    movel([0.070135, -1.347885, -2.596834, -0.767670, 1.570796, 1.640931],accel_mss,speed_ms,0,blend_radius_m)
    movel([0.070293, -1.348064, -2.596716, -0.767609, 1.570796, 1.641090],accel_mss,speed_ms,0,blend_radius_m)
    movel([0.070585, -1.348016, -2.596748, -0.767625, 1.570796, 1.641381],accel_mss,speed_ms,0,blend_radius_m)
    movel([0.071041, -1.347896, -2.596827, -0.767666, 1.570796, 1.641837],accel_mss,speed_ms,0,blend_radius_m)
    movel([0.071762, -1.347670, -2.596975, -0.767743, 1.570796, 1.642559],accel_mss,speed_ms,0,blend_radius_m)
    movel([0.072728, -1.347369, -2.597173, -0.767846, 1.570796, 1.643524],accel_mss,speed_ms,0,blend_radius_m)
    movel([0.073151, -1.347276, -2.597235, -0.767878, 1.570796, 1.643947],accel_mss,speed_ms,0,blend_radius_m)
    movel([0.073323, -1.347462, -2.597113, -0.767815, 1.570796, 1.644120],accel_mss,speed_ms,0,blend_radius_m)
    movel([0.072183, -1.349035, -2.596076, -0.767279, 1.570796, 1.642979],accel_mss,speed_ms,0,blend_radius_m)
    movel([0.070974, -1.350670, -2.594994, -0.766725, 1.570796, 1.641770],accel_mss,speed_ms,0,blend_radius_m)
    movel([0.069560, -1.352574, -2.593730, -0.766085, 1.570796, 1.640356],accel_mss,speed_ms,0,blend_radius_m)
    movel([0.068144, -1.354467, -2.592468, -0.765453, 1.570796, 1.638941],accel_mss,speed_ms,0,blend_radius_m)
    movel([0.066928, -1.356066, -2.591399, -0.764924, 1.570796, 1.637725],accel_mss,speed_ms,0,blend_radius_m)
    movel([0.065852, -1.357467, -2.590459, -0.764463, 1.570796, 1.636649],accel_mss,speed_ms,0,blend_radius_m)
    speed_ms = 0.003
    movel([0.065746, -1.344239, -2.584239, -0.783911, 1.570796, 1.636542],accel_mss,speed_ms,0,blend_radius_m)
    speed_ms = 1.000
    movel([0.065746, -1.318776, -2.571512, -0.822101, 1.570796, 1.636542],accel_mss,speed_ms,0,blend_radius_m)
    movel([0.081492, -1.289170, -2.589753, -0.833466, 1.570796, 1.652288],accel_mss,speed_ms,0,blend_radius_m)
    movel([0.081492, -1.315103, -2.602865, -0.794421, 1.570796, 1.652288],accel_mss,speed_ms,0,blend_radius_m)
    speed_ms = 0.003
    movel([0.081492, -1.325253, -2.607648, -0.779489, 1.570796, 1.652288],accel_mss,speed_ms,0,blend_radius_m)
    speed_ms = 0.007
    movel([0.081341, -1.325030, -2.607788, -0.779571, 1.570796, 1.652138],accel_mss,speed_ms,0,blend_radius_m)
    movel([0.081467, -1.324183, -2.608320, -0.779886, 1.570796, 1.652263],accel_mss,speed_ms,0,blend_radius_m)
    movel([0.081769, -1.322931, -2.609105, -0.780353, 1.570796, 1.652565],accel_mss,speed_ms,0,blend_radius_m)
    movel([0.082314, -1.321124, -2.610234, -0.781031, 1.570796, 1.653110],accel_mss,speed_ms,0,blend_radius_m)
    movel([0.082603, -1.320135, -2.610851, -0.781404, 1.570796, 1.653400],accel_mss,speed_ms,0,blend_radius_m)
    movel([0.082660, -1.319646, -2.611154, -0.781588, 1.570796, 1.653456],accel_mss,speed_ms,0,blend_radius_m)
    movel([0.082527, -1.319485, -2.611255, -0.781649, 1.570796, 1.653323],accel_mss,speed_ms,0,blend_radius_m)
    movel([0.082236, -1.319545, -2.611217, -0.781627, 1.570796, 1.653033],accel_mss,speed_ms,0,blend_radius_m)
    movel([0.081751, -1.319793, -2.611063, -0.781533, 1.570796, 1.652547],accel_mss,speed_ms,0,blend_radius_m)
    movel([0.081384, -1.319972, -2.610952, -0.781465, 1.570796, 1.652181],accel_mss,speed_ms,0,blend_radius_m)
    movel([0.081002, -1.320156, -2.610837, -0.781396, 1.570796, 1.651798],accel_mss,speed_ms,0,blend_radius_m)
    movel([0.080195, -1.320466, -2.610644, -0.781279, 1.570796, 1.650992],accel_mss,speed_ms,0,blend_radius_m)
    movel([0.079870, -1.320370, -2.610704, -0.781315, 1.570796, 1.650667],accel_mss,speed_ms,0,blend_radius_m)
    movel([0.079791, -1.319865, -2.611018, -0.781506, 1.570796, 1.650588],accel_mss,speed_ms,0,blend_radius_m)
    movel([0.079966, -1.317934, -2.612217, -0.782238, 1.570796, 1.650762],accel_mss,speed_ms,0,blend_radius_m)
    movel([0.080077, -1.316920, -2.612844, -0.782625, 1.570796, 1.650873],accel_mss,speed_ms,0,blend_radius_m)
    movel([0.080182, -1.316146, -2.613323, -0.782921, 1.570796, 1.650979],accel_mss,speed_ms,0,blend_radius_m)
    movel([0.080285, -1.315545, -2.613693, -0.783151, 1.570796, 1.651081],accel_mss,speed_ms,0,blend_radius_m)
    movel([0.080559, -1.315193, -2.613910, -0.783286, 1.570796, 1.651355],accel_mss,speed_ms,0,blend_radius_m)
    movel([0.080916, -1.314988, -2.614036, -0.783365, 1.570796, 1.651713],accel_mss,speed_ms,0,blend_radius_m)
    movel([0.081474, -1.314721, -2.614200, -0.783468, 1.570796, 1.652271],accel_mss,speed_ms,0,blend_radius_m)
    movel([0.082380, -1.314335, -2.614437, -0.783616, 1.570796, 1.653176],accel_mss,speed_ms,0,blend_radius_m)
    movel([0.083212, -1.314002, -2.614642, -0.783745, 1.570796, 1.654008],accel_mss,speed_ms,0,blend_radius_m)
    movel([0.083713, -1.313842, -2.614741, -0.783807, 1.570796, 1.654510],accel_mss,speed_ms,0,blend_radius_m)
    movel([0.084029, -1.313805, -2.614764, -0.783821, 1.570796, 1.654826],accel_mss,speed_ms,0,blend_radius_m)
    movel([0.084275, -1.313954, -2.614672, -0.783763, 1.570796, 1.655071],accel_mss,speed_ms,0,blend_radius_m)
    movel([0.084281, -1.314246, -2.614492, -0.783650, 1.570796, 1.655077],accel_mss,speed_ms,0,blend_radius_m)
    movel([0.084076, -1.314711, -2.614206, -0.783471, 1.570796, 1.654872],accel_mss,speed_ms,0,blend_radius_m)
    movel([0.083648, -1.315836, -2.613514, -0.783039, 1.570796, 1.654444],accel_mss,speed_ms,0,blend_radius_m)
    movel([0.083205, -1.317019, -2.612783, -0.782587, 1.570796, 1.654001],accel_mss,speed_ms,0,blend_radius_m)
    movel([0.083202, -1.317302, -2.612608, -0.782479, 1.570796, 1.653998],accel_mss,speed_ms,0,blend_radius_m)
    movel([0.083652, -1.317193, -2.612675, -0.782520, 1.570796, 1.654448],accel_mss,speed_ms,0,blend_radius_m)
    movel([0.084222, -1.316970, -2.612813, -0.782605, 1.570796, 1.655019],accel_mss,speed_ms,0,blend_radius_m)
    movel([0.084649, -1.316806, -2.612915, -0.782668, 1.570796, 1.655445],accel_mss,speed_ms,0,blend_radius_m)
    movel([0.085028, -1.316673, -2.612997, -0.782719, 1.570796, 1.655825],accel_mss,speed_ms,0,blend_radius_m)
    movel([0.085344, -1.316573, -2.613059, -0.782757, 1.570796, 1.656140],accel_mss,speed_ms,0,blend_radius_m)
    movel([0.085547, -1.316717, -2.612970, -0.782702, 1.570796, 1.656343],accel_mss,speed_ms,0,blend_radius_m)
    movel([0.085460, -1.317124, -2.612719, -0.782547, 1.570796, 1.656257],accel_mss,speed_ms,0,blend_radius_m)
    movel([0.084802, -1.318680, -2.611754, -0.781955, 1.570796, 1.655598],accel_mss,speed_ms,0,blend_radius_m)
    movel([0.084057, -1.320391, -2.610691, -0.781307, 1.570796, 1.654853],accel_mss,speed_ms,0,blend_radius_m)
    movel([0.083277, -1.322119, -2.609613, -0.780657, 1.570796, 1.654073],accel_mss,speed_ms,0,blend_radius_m)
    movel([0.082971, -1.322793, -2.609192, -0.780405, 1.570796, 1.653767],accel_mss,speed_ms,0,blend_radius_m)
    movel([0.082683, -1.323437, -2.608788, -0.780164, 1.570796, 1.653479],accel_mss,speed_ms,0,blend_radius_m)
    movel([0.082444, -1.323982, -2.608446, -0.779961, 1.570796, 1.653241],accel_mss,speed_ms,0,blend_radius_m)
    movel([0.082332, -1.324263, -2.608270, -0.779856, 1.570796, 1.653129],accel_mss,speed_ms,0,blend_radius_m)
    movel([0.082154, -1.324637, -2.608035, -0.779717, 1.570796, 1.652950],accel_mss,speed_ms,0,blend_radius_m)
    movel([0.081915, -1.324973, -2.607824, -0.779592, 1.570796, 1.652711],accel_mss,speed_ms,0,blend_radius_m)
    movel([0.081676, -1.325197, -2.607683, -0.779509, 1.570796, 1.652472],accel_mss,speed_ms,0,blend_radius_m)
    speed_ms = 0.003
    movel([0.081492, -1.328688, -2.609225, -0.774476, 1.570796, 1.652288],accel_mss,speed_ms,0,blend_radius_m)
    speed_ms = 0.007
    movel([0.081341, -1.328466, -2.609366, -0.774557, 1.570796, 1.652138],accel_mss,speed_ms,0,blend_radius_m)
    movel([0.081467, -1.327621, -2.609900, -0.774869, 1.570796, 1.652263],accel_mss,speed_ms,0,blend_radius_m)
    movel([0.081769, -1.326371, -2.610687, -0.775331, 1.570796, 1.652565],accel_mss,speed_ms,0,blend_radius_m)
    movel([0.082314, -1.324569, -2.611819, -0.776001, 1.570796, 1.653110],accel_mss,speed_ms,0,blend_radius_m)
    movel([0.082603, -1.323582, -2.612437, -0.776370, 1.570796, 1.653400],accel_mss,speed_ms,0,blend_radius_m)
    movel([0.082660, -1.323095, -2.612741, -0.776553, 1.570796, 1.653456],accel_mss,speed_ms,0,blend_radius_m)
    movel([0.082527, -1.322934, -2.612842, -0.776613, 1.570796, 1.653323],accel_mss,speed_ms,0,blend_radius_m)
    movel([0.082236, -1.322994, -2.612804, -0.776590, 1.570796, 1.653033],accel_mss,speed_ms,0,blend_radius_m)
    movel([0.081751, -1.323241, -2.612650, -0.776498, 1.570796, 1.652547],accel_mss,speed_ms,0,blend_radius_m)
    movel([0.081384, -1.323420, -2.612538, -0.776431, 1.570796, 1.652181],accel_mss,speed_ms,0,blend_radius_m)
    movel([0.081002, -1.323604, -2.612423, -0.776362, 1.570796, 1.651798],accel_mss,speed_ms,0,blend_radius_m)
    movel([0.080195, -1.323913, -2.612230, -0.776246, 1.570796, 1.650992],accel_mss,speed_ms,0,blend_radius_m)
    movel([0.079870, -1.323817, -2.612290, -0.776282, 1.570796, 1.650667],accel_mss,speed_ms,0,blend_radius_m)
    movel([0.079791, -1.323313, -2.612605, -0.776471, 1.570796, 1.650588],accel_mss,speed_ms,0,blend_radius_m)
    movel([0.079966, -1.321386, -2.613807, -0.777196, 1.570796, 1.650762],accel_mss,speed_ms,0,blend_radius_m)
    movel([0.080077, -1.320375, -2.614436, -0.777578, 1.570796, 1.650873],accel_mss,speed_ms,0,blend_radius_m)
    movel([0.080182, -1.319602, -2.614916, -0.777871, 1.570796, 1.650979],accel_mss,speed_ms,0,blend_radius_m)
    movel([0.080285, -1.319004, -2.615287, -0.778098, 1.570796, 1.651081],accel_mss,speed_ms,0,blend_radius_m)
    movel([0.080559, -1.318652, -2.615504, -0.778232, 1.570796, 1.651355],accel_mss,speed_ms,0,blend_radius_m)
    movel([0.080916, -1.318448, -2.615631, -0.778310, 1.570796, 1.651713],accel_mss,speed_ms,0,blend_radius_m)
    movel([0.081474, -1.318181, -2.615796, -0.778412, 1.570796, 1.652271],accel_mss,speed_ms,0,blend_radius_m)
    movel([0.082380, -1.317797, -2.616034, -0.778559, 1.570796, 1.653176],accel_mss,speed_ms,0,blend_radius_m)
    movel([0.083212, -1.317464, -2.616239, -0.778686, 1.570796, 1.654008],accel_mss,speed_ms,0,blend_radius_m)
    movel([0.083713, -1.317304, -2.616338, -0.778747, 1.570796, 1.654510],accel_mss,speed_ms,0,blend_radius_m)
    movel([0.084029, -1.317267, -2.616361, -0.778761, 1.570796, 1.654826],accel_mss,speed_ms,0,blend_radius_m)
    movel([0.084275, -1.317416, -2.616269, -0.778704, 1.570796, 1.655071],accel_mss,speed_ms,0,blend_radius_m)
    movel([0.084281, -1.317708, -2.616088, -0.778593, 1.570796, 1.655077],accel_mss,speed_ms,0,blend_radius_m)
    movel([0.084076, -1.318171, -2.615802, -0.778416, 1.570796, 1.654872],accel_mss,speed_ms,0,blend_radius_m)
    movel([0.083648, -1.319294, -2.615107, -0.777988, 1.570796, 1.654444],accel_mss,speed_ms,0,blend_radius_m)
    movel([0.083205, -1.320474, -2.614375, -0.777540, 1.570796, 1.654001],accel_mss,speed_ms,0,blend_radius_m)
    movel([0.083202, -1.320756, -2.614200, -0.777434, 1.570796, 1.653998],accel_mss,speed_ms,0,blend_radius_m)
    movel([0.083652, -1.320648, -2.614267, -0.777475, 1.570796, 1.654448],accel_mss,speed_ms,0,blend_radius_m)
    movel([0.084222, -1.320425, -2.614405, -0.777559, 1.570796, 1.655019],accel_mss,speed_ms,0,blend_radius_m)
    movel([0.084649, -1.320261, -2.614507, -0.777621, 1.570796, 1.655445],accel_mss,speed_ms,0,blend_radius_m)
    movel([0.085028, -1.320129, -2.614589, -0.777671, 1.570796, 1.655825],accel_mss,speed_ms,0,blend_radius_m)
    movel([0.085344, -1.320029, -2.614651, -0.777709, 1.570796, 1.656140],accel_mss,speed_ms,0,blend_radius_m)
    movel([0.085547, -1.320173, -2.614562, -0.777654, 1.570796, 1.656343],accel_mss,speed_ms,0,blend_radius_m)
    movel([0.085460, -1.320578, -2.614310, -0.777501, 1.570796, 1.656257],accel_mss,speed_ms,0,blend_radius_m)
    movel([0.084802, -1.322131, -2.613343, -0.776915, 1.570796, 1.655598],accel_mss,speed_ms,0,blend_radius_m)
    movel([0.084057, -1.323838, -2.612277, -0.776274, 1.570796, 1.654853],accel_mss,speed_ms,0,blend_radius_m)
    movel([0.083277, -1.325561, -2.611196, -0.775632, 1.570796, 1.654073],accel_mss,speed_ms,0,blend_radius_m)
    movel([0.082971, -1.326234, -2.610773, -0.775382, 1.570796, 1.653767],accel_mss,speed_ms,0,blend_radius_m)
    movel([0.082683, -1.326877, -2.610369, -0.775144, 1.570796, 1.653479],accel_mss,speed_ms,0,blend_radius_m)
    movel([0.082444, -1.327420, -2.610026, -0.774943, 1.570796, 1.653241],accel_mss,speed_ms,0,blend_radius_m)
    movel([0.082332, -1.327700, -2.609849, -0.774839, 1.570796, 1.653129],accel_mss,speed_ms,0,blend_radius_m)
    movel([0.082154, -1.328074, -2.609613, -0.774702, 1.570796, 1.652950],accel_mss,speed_ms,0,blend_radius_m)
    movel([0.081915, -1.328409, -2.609402, -0.774578, 1.570796, 1.652711],accel_mss,speed_ms,0,blend_radius_m)
    movel([0.081676, -1.328633, -2.609260, -0.774496, 1.570796, 1.652472],accel_mss,speed_ms,0,blend_radius_m)
    speed_ms = 0.003
    movel([0.081492, -1.315103, -2.602865, -0.794421, 1.570796, 1.652288],accel_mss,speed_ms,0,blend_radius_m)
    speed_ms = 1.000
    movel([0.081492, -1.289170, -2.589753, -0.833466, 1.570796, 1.652288],accel_mss,speed_ms,0,blend_radius_m)
    movel([0.084778, -1.290377, -2.589031, -0.832981, 1.570796, 1.655574],accel_mss,speed_ms,0,blend_radius_m)
    movel([0.084778, -1.316292, -2.602127, -0.793970, 1.570796, 1.655574],accel_mss,speed_ms,0,blend_radius_m)
    speed_ms = 0.003
    movel([0.084778, -1.326433, -2.606904, -0.779052, 1.570796, 1.655574],accel_mss,speed_ms,0,blend_radius_m)
    speed_ms = 0.007
    movel([0.090842, -1.323774, -2.608577, -0.780038, 1.570796, 1.661638],accel_mss,speed_ms,0,blend_radius_m)
    movel([0.097024, -1.321322, -2.610111, -0.780956, 1.570796, 1.667820],accel_mss,speed_ms,0,blend_radius_m)
    movel([0.098922, -1.320620, -2.610549, -0.781221, 1.570796, 1.669718],accel_mss,speed_ms,0,blend_radius_m)
    movel([0.099688, -1.320397, -2.610687, -0.781305, 1.570796, 1.670484],accel_mss,speed_ms,0,blend_radius_m)
    movel([0.100116, -1.320391, -2.610691, -0.781307, 1.570796, 1.670912],accel_mss,speed_ms,0,blend_radius_m)
    movel([0.100432, -1.320571, -2.610579, -0.781239, 1.570796, 1.671229],accel_mss,speed_ms,0,blend_radius_m)
    movel([0.100558, -1.320745, -2.610471, -0.781174, 1.570796, 1.671354],accel_mss,speed_ms,0,blend_radius_m)
    movel([0.100527, -1.321057, -2.610276, -0.781056, 1.570796, 1.671323],accel_mss,speed_ms,0,blend_radius_m)
    movel([0.100222, -1.321346, -2.610096, -0.780947, 1.570796, 1.671018],accel_mss,speed_ms,0,blend_radius_m)
    movel([0.099520, -1.321694, -2.609879, -0.780817, 1.570796, 1.670316],accel_mss,speed_ms,0,blend_radius_m)
    movel([0.098688, -1.322091, -2.609630, -0.780668, 1.570796, 1.669485],accel_mss,speed_ms,0,blend_radius_m)
    movel([0.097742, -1.322527, -2.609358, -0.780504, 1.570796, 1.668538],accel_mss,speed_ms,0,blend_radius_m)
    movel([0.096707, -1.322998, -2.609063, -0.780328, 1.570796, 1.667503],accel_mss,speed_ms,0,blend_radius_m)
    movel([0.095604, -1.323499, -2.608749, -0.780141, 1.570796, 1.666400],accel_mss,speed_ms,0,blend_radius_m)
    movel([0.094597, -1.323965, -2.608457, -0.779967, 1.570796, 1.665393],accel_mss,speed_ms,0,blend_radius_m)
    movel([0.093881, -1.324296, -2.608249, -0.779844, 1.570796, 1.664677],accel_mss,speed_ms,0,blend_radius_m)
    movel([0.092978, -1.324716, -2.607985, -0.779688, 1.570796, 1.663774],accel_mss,speed_ms,0,blend_radius_m)
    movel([0.090797, -1.325723, -2.607352, -0.779314, 1.570796, 1.661593],accel_mss,speed_ms,0,blend_radius_m)
    movel([0.088204, -1.326921, -2.606596, -0.778872, 1.570796, 1.659000],accel_mss,speed_ms,0,blend_radius_m)
    movel([0.085405, -1.328216, -2.605777, -0.778396, 1.570796, 1.656201],accel_mss,speed_ms,0,blend_radius_m)
    movel([0.082317, -1.329650, -2.604868, -0.777871, 1.570796, 1.653113],accel_mss,speed_ms,0,blend_radius_m)
    movel([0.078847, -1.331268, -2.603839, -0.777282, 1.570796, 1.649643],accel_mss,speed_ms,0,blend_radius_m)
    movel([0.075532, -1.332819, -2.602849, -0.776722, 1.570796, 1.646329],accel_mss,speed_ms,0,blend_radius_m)
    movel([0.072957, -1.334028, -2.602074, -0.776286, 1.570796, 1.643754],accel_mss,speed_ms,0,blend_radius_m)
    movel([0.070326, -1.335262, -2.601283, -0.775845, 1.570796, 1.641122],accel_mss,speed_ms,0,blend_radius_m)
    movel([0.068708, -1.336000, -2.600808, -0.775581, 1.570796, 1.639505],accel_mss,speed_ms,0,blend_radius_m)
    movel([0.067572, -1.336501, -2.600485, -0.775403, 1.570796, 1.638368],accel_mss,speed_ms,0,blend_radius_m)
    movel([0.067250, -1.336369, -2.600570, -0.775450, 1.570796, 1.638047],accel_mss,speed_ms,0,blend_radius_m)
    movel([0.067250, -1.336102, -2.600742, -0.775545, 1.570796, 1.638047],accel_mss,speed_ms,0,blend_radius_m)
    movel([0.067376, -1.335776, -2.600952, -0.775661, 1.570796, 1.638173],accel_mss,speed_ms,0,blend_radius_m)
    movel([0.067604, -1.335465, -2.601152, -0.775772, 1.570796, 1.638401],accel_mss,speed_ms,0,blend_radius_m)
    movel([0.067983, -1.335141, -2.601360, -0.775888, 1.570796, 1.638779],accel_mss,speed_ms,0,blend_radius_m)
    movel([0.068669, -1.334712, -2.601636, -0.776041, 1.570796, 1.639465],accel_mss,speed_ms,0,blend_radius_m)
    movel([0.069880, -1.334026, -2.602076, -0.776287, 1.570796, 1.640676],accel_mss,speed_ms,0,blend_radius_m)
    movel([0.072622, -1.332531, -2.603033, -0.776825, 1.570796, 1.643418],accel_mss,speed_ms,0,blend_radius_m)
    movel([0.078735, -1.329339, -2.605065, -0.777984, 1.570796, 1.649532],accel_mss,speed_ms,0,blend_radius_m)
    movel([0.084778, -1.326433, -2.606904, -0.779052, 1.570796, 1.655574],accel_mss,speed_ms,0,blend_radius_m)
    speed_ms = 0.003
    movel([0.084778, -1.329866, -2.608480, -0.774044, 1.570796, 1.655574],accel_mss,speed_ms,0,blend_radius_m)
    speed_ms = 0.007
    movel([0.090842, -1.327213, -2.610157, -0.775019, 1.570796, 1.661638],accel_mss,speed_ms,0,blend_radius_m)
    movel([0.097024, -1.324766, -2.611695, -0.775928, 1.570796, 1.667820],accel_mss,speed_ms,0,blend_radius_m)
    movel([0.098922, -1.324066, -2.612134, -0.776189, 1.570796, 1.669718],accel_mss,speed_ms,0,blend_radius_m)
    movel([0.099688, -1.323844, -2.612273, -0.776272, 1.570796, 1.670484],accel_mss,speed_ms,0,blend_radius_m)
    movel([0.100116, -1.323838, -2.612277, -0.776274, 1.570796, 1.670912],accel_mss,speed_ms,0,blend_radius_m)
    movel([0.100432, -1.324018, -2.612164, -0.776207, 1.570796, 1.671229],accel_mss,speed_ms,0,blend_radius_m)
    movel([0.100558, -1.324191, -2.612056, -0.776142, 1.570796, 1.671354],accel_mss,speed_ms,0,blend_radius_m)
    movel([0.100527, -1.324503, -2.611860, -0.776026, 1.570796, 1.671323],accel_mss,speed_ms,0,blend_radius_m)
    movel([0.100222, -1.324790, -2.611680, -0.775919, 1.570796, 1.671018],accel_mss,speed_ms,0,blend_radius_m)
    movel([0.099520, -1.325137, -2.611462, -0.775789, 1.570796, 1.670316],accel_mss,speed_ms,0,blend_radius_m)
    movel([0.098688, -1.325534, -2.611213, -0.775642, 1.570796, 1.669485],accel_mss,speed_ms,0,blend_radius_m)
    movel([0.097742, -1.325969, -2.610940, -0.775480, 1.570796, 1.668538],accel_mss,speed_ms,0,blend_radius_m)
    movel([0.096707, -1.326438, -2.610645, -0.775306, 1.570796, 1.667503],accel_mss,speed_ms,0,blend_radius_m)
    movel([0.095604, -1.326939, -2.610330, -0.775121, 1.570796, 1.666400],accel_mss,speed_ms,0,blend_radius_m)
    movel([0.094597, -1.327403, -2.610037, -0.774949, 1.570796, 1.665393],accel_mss,speed_ms,0,blend_radius_m)
    movel([0.093881, -1.327733, -2.609828, -0.774827, 1.570796, 1.664677],accel_mss,speed_ms,0,blend_radius_m)
    movel([0.092978, -1.328152, -2.609564, -0.774673, 1.570796, 1.663774],accel_mss,speed_ms,0,blend_radius_m)
    movel([0.090797, -1.329157, -2.608929, -0.774303, 1.570796, 1.661593],accel_mss,speed_ms,0,blend_radius_m)
    movel([0.088204, -1.330352, -2.608171, -0.773866, 1.570796, 1.659000],accel_mss,speed_ms,0,blend_radius_m)
    movel([0.085405, -1.331644, -2.607350, -0.773395, 1.570796, 1.656201],accel_mss,speed_ms,0,blend_radius_m)
    movel([0.082317, -1.333074, -2.606438, -0.772876, 1.570796, 1.653113],accel_mss,speed_ms,0,blend_radius_m)
    movel([0.078847, -1.334688, -2.605406, -0.772294, 1.570796, 1.649643],accel_mss,speed_ms,0,blend_radius_m)
    movel([0.075532, -1.336235, -2.604414, -0.771740, 1.570796, 1.646329],accel_mss,speed_ms,0,blend_radius_m)
    movel([0.072957, -1.337442, -2.603637, -0.771310, 1.570796, 1.643754],accel_mss,speed_ms,0,blend_radius_m)
    movel([0.070326, -1.338672, -2.602844, -0.770873, 1.570796, 1.641122],accel_mss,speed_ms,0,blend_radius_m)
    movel([0.068708, -1.339409, -2.602367, -0.770613, 1.570796, 1.639505],accel_mss,speed_ms,0,blend_radius_m)
    movel([0.067572, -1.339908, -2.602044, -0.770437, 1.570796, 1.638368],accel_mss,speed_ms,0,blend_radius_m)
    movel([0.067250, -1.339777, -2.602129, -0.770483, 1.570796, 1.638047],accel_mss,speed_ms,0,blend_radius_m)
    movel([0.067250, -1.339511, -2.602301, -0.770577, 1.570796, 1.638047],accel_mss,speed_ms,0,blend_radius_m)
    movel([0.067376, -1.339185, -2.602512, -0.770692, 1.570796, 1.638173],accel_mss,speed_ms,0,blend_radius_m)
    movel([0.067604, -1.338875, -2.602713, -0.770802, 1.570796, 1.638401],accel_mss,speed_ms,0,blend_radius_m)
    movel([0.067983, -1.338552, -2.602921, -0.770916, 1.570796, 1.638779],accel_mss,speed_ms,0,blend_radius_m)
    movel([0.068669, -1.338124, -2.603197, -0.771067, 1.570796, 1.639465],accel_mss,speed_ms,0,blend_radius_m)
    movel([0.069880, -1.337439, -2.603639, -0.771311, 1.570796, 1.640676],accel_mss,speed_ms,0,blend_radius_m)
    movel([0.072622, -1.335949, -2.604598, -0.771843, 1.570796, 1.643418],accel_mss,speed_ms,0,blend_radius_m)
    movel([0.078735, -1.332764, -2.606636, -0.772988, 1.570796, 1.649532],accel_mss,speed_ms,0,blend_radius_m)
    movel([0.084778, -1.329866, -2.608480, -0.774044, 1.570796, 1.655574],accel_mss,speed_ms,0,blend_radius_m)
    speed_ms = 0.003
    movel([0.084778, -1.316292, -2.602127, -0.793970, 1.570796, 1.655574],accel_mss,speed_ms,0,blend_radius_m)
    speed_ms = 1.000
    movel([0.084778, -1.290377, -2.589031, -0.832981, 1.570796, 1.655574],accel_mss,speed_ms,0,blend_radius_m)
    movel([0.084148, -1.290304, -2.589074, -0.833010, 1.570796, 1.654945],accel_mss,speed_ms,0,blend_radius_m)
    movel([0.084148, -1.316221, -2.602171, -0.793997, 1.570796, 1.654945],accel_mss,speed_ms,0,blend_radius_m)
    speed_ms = 0.003
    movel([0.084148, -1.326362, -2.606949, -0.779078, 1.570796, 1.654945],accel_mss,speed_ms,0,blend_radius_m)
    speed_ms = 0.007
    movel([0.080371, -1.328162, -2.605812, -0.778416, 1.570796, 1.651168],accel_mss,speed_ms,0,blend_radius_m)
    movel([0.077408, -1.329664, -2.604859, -0.777866, 1.570796, 1.648205],accel_mss,speed_ms,0,blend_radius_m)
    movel([0.073168, -1.331900, -2.603435, -0.777053, 1.570796, 1.643964],accel_mss,speed_ms,0,blend_radius_m)
    movel([0.068676, -1.334302, -2.601899, -0.776188, 1.570796, 1.639472],accel_mss,speed_ms,0,blend_radius_m)
    movel([0.068123, -1.334676, -2.601659, -0.776054, 1.570796, 1.638919],accel_mss,speed_ms,0,blend_radius_m)
    movel([0.067836, -1.334677, -2.601658, -0.776054, 1.570796, 1.638633],accel_mss,speed_ms,0,blend_radius_m)
    movel([0.067589, -1.333691, -2.602291, -0.776408, 1.570796, 1.638385],accel_mss,speed_ms,0,blend_radius_m)
    movel([0.067346, -1.332066, -2.603330, -0.776993, 1.570796, 1.638142],accel_mss,speed_ms,0,blend_radius_m)
    movel([0.067096, -1.329414, -2.605018, -0.777957, 1.570796, 1.637892],accel_mss,speed_ms,0,blend_radius_m)
    movel([0.067029, -1.326857, -2.606636, -0.778895, 1.570796, 1.637826],accel_mss,speed_ms,0,blend_radius_m)
    movel([0.067221, -1.323815, -2.608551, -0.780023, 1.570796, 1.638017],accel_mss,speed_ms,0,blend_radius_m)
    movel([0.067565, -1.320910, -2.610368, -0.781111, 1.570796, 1.638361],accel_mss,speed_ms,0,blend_radius_m)
    movel([0.068023, -1.319911, -2.610990, -0.781488, 1.570796, 1.638820],accel_mss,speed_ms,0,blend_radius_m)
    movel([0.068550, -1.319416, -2.611298, -0.781676, 1.570796, 1.639347],accel_mss,speed_ms,0,blend_radius_m)
    movel([0.070937, -1.317784, -2.612310, -0.782295, 1.570796, 1.641733],accel_mss,speed_ms,0,blend_radius_m)
    movel([0.073484, -1.316103, -2.613349, -0.782937, 1.570796, 1.644281],accel_mss,speed_ms,0,blend_radius_m)
    movel([0.075813, -1.314653, -2.614242, -0.783494, 1.570796, 1.646609],accel_mss,speed_ms,0,blend_radius_m)
    movel([0.078779, -1.312938, -2.615295, -0.784156, 1.570796, 1.649576],accel_mss,speed_ms,0,blend_radius_m)
    movel([0.081413, -1.311574, -2.616130, -0.784685, 1.570796, 1.652209],accel_mss,speed_ms,0,blend_radius_m)
    movel([0.084118, -1.310360, -2.616871, -0.785158, 1.570796, 1.654915],accel_mss,speed_ms,0,blend_radius_m)
    movel([0.087305, -1.309106, -2.617634, -0.785649, 1.570796, 1.658101],accel_mss,speed_ms,0,blend_radius_m)
    movel([0.089778, -1.308243, -2.618158, -0.785988, 1.570796, 1.660575],accel_mss,speed_ms,0,blend_radius_m)
    movel([0.092672, -1.307345, -2.618702, -0.786342, 1.570796, 1.663468],accel_mss,speed_ms,0,blend_radius_m)
    movel([0.095427, -1.306558, -2.619178, -0.786653, 1.570796, 1.666223],accel_mss,speed_ms,0,blend_radius_m)
    movel([0.096203, -1.306481, -2.619225, -0.786683, 1.570796, 1.666999],accel_mss,speed_ms,0,blend_radius_m)
    movel([0.096612, -1.306789, -2.619039, -0.786561, 1.570796, 1.667408],accel_mss,speed_ms,0,blend_radius_m)
    movel([0.096874, -1.307161, -2.618814, -0.786415, 1.570796, 1.667670],accel_mss,speed_ms,0,blend_radius_m)
    movel([0.097202, -1.307715, -2.618478, -0.786196, 1.570796, 1.667998],accel_mss,speed_ms,0,blend_radius_m)
    movel([0.098014, -1.309498, -2.617396, -0.785496, 1.570796, 1.668810],accel_mss,speed_ms,0,blend_radius_m)
    movel([0.098672, -1.311674, -2.616069, -0.784646, 1.570796, 1.669469],accel_mss,speed_ms,0,blend_radius_m)
    movel([0.099188, -1.314269, -2.614478, -0.783642, 1.570796, 1.669984],accel_mss,speed_ms,0,blend_radius_m)
    movel([0.099569, -1.317326, -2.612593, -0.782470, 1.570796, 1.670365],accel_mss,speed_ms,0,blend_radius_m)
    movel([0.099684, -1.318625, -2.611789, -0.781975, 1.570796, 1.670481],accel_mss,speed_ms,0,blend_radius_m)
    movel([0.099703, -1.319328, -2.611352, -0.781709, 1.570796, 1.670499],accel_mss,speed_ms,0,blend_radius_m)
    movel([0.099661, -1.319764, -2.611081, -0.781544, 1.570796, 1.670458],accel_mss,speed_ms,0,blend_radius_m)
    movel([0.099398, -1.320054, -2.610901, -0.781434, 1.570796, 1.670194],accel_mss,speed_ms,0,blend_radius_m)
    movel([0.098670, -1.320347, -2.610718, -0.781324, 1.570796, 1.669466],accel_mss,speed_ms,0,blend_radius_m)
    movel([0.097818, -1.320681, -2.610510, -0.781198, 1.570796, 1.668615],accel_mss,speed_ms,0,blend_radius_m)
    movel([0.096841, -1.321053, -2.610278, -0.781057, 1.570796, 1.667638],accel_mss,speed_ms,0,blend_radius_m)
    movel([0.092668, -1.322683, -2.609260, -0.780446, 1.570796, 1.663465],accel_mss,speed_ms,0,blend_radius_m)
    movel([0.088344, -1.324493, -2.608126, -0.779771, 1.570796, 1.659140],accel_mss,speed_ms,0,blend_radius_m)
    movel([0.084148, -1.326362, -2.606949, -0.779078, 1.570796, 1.654945],accel_mss,speed_ms,0,blend_radius_m)
    speed_ms = 0.003
    movel([0.084148, -1.329795, -2.608525, -0.774070, 1.570796, 1.654945],accel_mss,speed_ms,0,blend_radius_m)
    speed_ms = 0.007
    movel([0.080371, -1.331590, -2.607385, -0.773415, 1.570796, 1.651168],accel_mss,speed_ms,0,blend_radius_m)
    movel([0.077408, -1.333089, -2.606429, -0.772871, 1.570796, 1.648205],accel_mss,speed_ms,0,blend_radius_m)
    movel([0.073168, -1.335319, -2.605002, -0.772068, 1.570796, 1.643964],accel_mss,speed_ms,0,blend_radius_m)
    movel([0.068676, -1.337715, -2.603461, -0.771213, 1.570796, 1.639472],accel_mss,speed_ms,0,blend_radius_m)
    movel([0.068123, -1.338088, -2.603221, -0.771080, 1.570796, 1.638919],accel_mss,speed_ms,0,blend_radius_m)
    movel([0.067836, -1.338089, -2.603220, -0.771080, 1.570796, 1.638633],accel_mss,speed_ms,0,blend_radius_m)
    movel([0.067589, -1.337105, -2.603854, -0.771430, 1.570796, 1.638385],accel_mss,speed_ms,0,blend_radius_m)
    movel([0.067346, -1.335484, -2.604896, -0.772009, 1.570796, 1.638142],accel_mss,speed_ms,0,blend_radius_m)
    movel([0.067096, -1.332839, -2.606589, -0.772962, 1.570796, 1.637892],accel_mss,speed_ms,0,blend_radius_m)
    movel([0.067029, -1.330288, -2.608211, -0.773889, 1.570796, 1.637826],accel_mss,speed_ms,0,blend_radius_m)
    movel([0.067221, -1.327253, -2.610131, -0.775004, 1.570796, 1.638017],accel_mss,speed_ms,0,blend_radius_m)
    movel([0.067565, -1.324356, -2.611953, -0.776081, 1.570796, 1.638361],accel_mss,speed_ms,0,blend_radius_m)
    movel([0.068023, -1.323359, -2.612577, -0.776454, 1.570796, 1.638820],accel_mss,speed_ms,0,blend_radius_m)
    movel([0.068550, -1.322865, -2.612885, -0.776639, 1.570796, 1.639347],accel_mss,speed_ms,0,blend_radius_m)
    movel([0.070937, -1.321237, -2.613900, -0.777252, 1.570796, 1.641733],accel_mss,speed_ms,0,blend_radius_m)
    movel([0.073484, -1.319560, -2.614942, -0.777887, 1.570796, 1.644281],accel_mss,speed_ms,0,blend_radius_m)
    movel([0.075813, -1.318113, -2.615838, -0.778438, 1.570796, 1.646609],accel_mss,speed_ms,0,blend_radius_m)
    movel([0.078779, -1.316403, -2.616894, -0.779093, 1.570796, 1.649576],accel_mss,speed_ms,0,blend_radius_m)
    movel([0.081413, -1.315042, -2.617730, -0.779617, 1.570796, 1.652209],accel_mss,speed_ms,0,blend_radius_m)
    movel([0.084118, -1.313831, -2.618473, -0.780085, 1.570796, 1.654915],accel_mss,speed_ms,0,blend_radius_m)
    movel([0.087305, -1.312579, -2.619239, -0.780571, 1.570796, 1.658101],accel_mss,speed_ms,0,blend_radius_m)
    movel([0.089778, -1.311718, -2.619764, -0.780906, 1.570796, 1.660575],accel_mss,speed_ms,0,blend_radius_m)
    movel([0.092672, -1.310823, -2.620310, -0.781256, 1.570796, 1.663468],accel_mss,speed_ms,0,blend_radius_m)
    movel([0.095427, -1.310038, -2.620787, -0.781564, 1.570796, 1.666223],accel_mss,speed_ms,0,blend_radius_m)
    movel([0.096203, -1.309960, -2.620834, -0.781594, 1.570796, 1.666999],accel_mss,speed_ms,0,blend_radius_m)
    movel([0.096612, -1.310268, -2.620648, -0.781474, 1.570796, 1.667408],accel_mss,speed_ms,0,blend_radius_m)
    movel([0.096874, -1.310638, -2.620422, -0.781328, 1.570796, 1.667670],accel_mss,speed_ms,0,blend_radius_m)
    movel([0.097202, -1.311192, -2.620085, -0.781112, 1.570796, 1.667998],accel_mss,speed_ms,0,blend_radius_m)
    movel([0.098014, -1.312970, -2.619000, -0.780419, 1.570796, 1.668810],accel_mss,speed_ms,0,blend_radius_m)
    movel([0.098672, -1.315142, -2.617669, -0.779578, 1.570796, 1.669469],accel_mss,speed_ms,0,blend_radius_m)
    movel([0.099188, -1.317731, -2.616074, -0.778584, 1.570796, 1.669984],accel_mss,speed_ms,0,blend_radius_m)
    movel([0.099569, -1.320780, -2.614184, -0.777424, 1.570796, 1.670365],accel_mss,speed_ms,0,blend_radius_m)
    movel([0.099684, -1.322076, -2.613377, -0.776935, 1.570796, 1.670481],accel_mss,speed_ms,0,blend_radius_m)
    movel([0.099703, -1.322777, -2.612940, -0.776672, 1.570796, 1.670499],accel_mss,speed_ms,0,blend_radius_m)
    movel([0.099661, -1.323212, -2.612668, -0.776509, 1.570796, 1.670458],accel_mss,speed_ms,0,blend_radius_m)
    movel([0.099398, -1.323501, -2.612487, -0.776400, 1.570796, 1.670194],accel_mss,speed_ms,0,blend_radius_m)
    movel([0.098670, -1.323794, -2.612304, -0.776291, 1.570796, 1.669466],accel_mss,speed_ms,0,blend_radius_m)
    movel([0.097818, -1.324127, -2.612096, -0.776166, 1.570796, 1.668615],accel_mss,speed_ms,0,blend_radius_m)
    movel([0.096841, -1.324498, -2.611863, -0.776027, 1.570796, 1.667638],accel_mss,speed_ms,0,blend_radius_m)
    movel([0.092668, -1.326124, -2.610842, -0.775423, 1.570796, 1.663465],accel_mss,speed_ms,0,blend_radius_m)
    movel([0.088344, -1.327930, -2.609704, -0.774755, 1.570796, 1.659140],accel_mss,speed_ms,0,blend_radius_m)
    movel([0.084148, -1.329795, -2.608525, -0.774070, 1.570796, 1.654945],accel_mss,speed_ms,0,blend_radius_m)
    speed_ms = 0.003
    movel([0.084148, -1.316221, -2.602171, -0.793997, 1.570796, 1.654945],accel_mss,speed_ms,0,blend_radius_m)
    speed_ms = 1.000
    movel([0.084148, -1.290304, -2.589074, -0.833010, 1.570796, 1.654945],accel_mss,speed_ms,0,blend_radius_m)
    movel([0.103618, -1.282197, -2.593889, -0.836303, 1.570796, 1.674414],accel_mss,speed_ms,0,blend_radius_m)
    movel([0.103618, -1.308235, -2.607092, -0.797062, 1.570796, 1.674414],accel_mss,speed_ms,0,blend_radius_m)
    speed_ms = 0.003
    movel([0.103618, -1.318431, -2.611909, -0.782049, 1.570796, 1.674414],accel_mss,speed_ms,0,blend_radius_m)
    speed_ms = 0.007
    movel([0.103637, -1.318157, -2.612079, -0.782153, 1.570796, 1.674433],accel_mss,speed_ms,0,blend_radius_m)
    movel([0.103885, -1.317021, -2.612782, -0.782586, 1.570796, 1.674681],accel_mss,speed_ms,0,blend_radius_m)
    movel([0.104417, -1.315534, -2.613700, -0.783155, 1.570796, 1.675214],accel_mss,speed_ms,0,blend_radius_m)
    movel([0.105039, -1.314112, -2.614575, -0.783702, 1.570796, 1.675836],accel_mss,speed_ms,0,blend_radius_m)
    movel([0.105483, -1.313585, -2.614898, -0.783906, 1.570796, 1.676279],accel_mss,speed_ms,0,blend_radius_m)
    movel([0.105791, -1.313406, -2.615008, -0.783975, 1.570796, 1.676587],accel_mss,speed_ms,0,blend_radius_m)
    movel([0.106222, -1.313247, -2.615105, -0.784036, 1.570796, 1.677018],accel_mss,speed_ms,0,blend_radius_m)
    movel([0.106665, -1.313136, -2.615174, -0.784079, 1.570796, 1.677462],accel_mss,speed_ms,0,blend_radius_m)
    movel([0.107028, -1.313106, -2.615192, -0.784091, 1.570796, 1.677825],accel_mss,speed_ms,0,blend_radius_m)
    movel([0.107242, -1.313211, -2.615128, -0.784050, 1.570796, 1.678039],accel_mss,speed_ms,0,blend_radius_m)
    movel([0.107306, -1.313480, -2.614963, -0.783946, 1.570796, 1.678102],accel_mss,speed_ms,0,blend_radius_m)
    movel([0.107218, -1.314076, -2.614597, -0.783716, 1.570796, 1.678014],accel_mss,speed_ms,0,blend_radius_m)
    movel([0.106840, -1.315758, -2.613562, -0.783069, 1.570796, 1.677636],accel_mss,speed_ms,0,blend_radius_m)
    movel([0.106420, -1.317549, -2.612455, -0.782385, 1.570796, 1.677217],accel_mss,speed_ms,0,blend_radius_m)
    movel([0.106260, -1.318107, -2.612110, -0.782172, 1.570796, 1.677056],accel_mss,speed_ms,0,blend_radius_m)
    movel([0.106100, -1.318394, -2.611932, -0.782063, 1.570796, 1.676897],accel_mss,speed_ms,0,blend_radius_m)
    movel([0.105428, -1.318749, -2.611711, -0.781928, 1.570796, 1.676224],accel_mss,speed_ms,0,blend_radius_m)
    movel([0.104756, -1.318864, -2.611640, -0.781885, 1.570796, 1.675553],accel_mss,speed_ms,0,blend_radius_m)
    movel([0.104107, -1.318923, -2.611604, -0.781862, 1.570796, 1.674903],accel_mss,speed_ms,0,blend_radius_m)
    movel([0.103793, -1.318857, -2.611645, -0.781887, 1.570796, 1.674589],accel_mss,speed_ms,0,blend_radius_m)
    movel([0.103635, -1.318631, -2.611785, -0.781973, 1.570796, 1.674432],accel_mss,speed_ms,0,blend_radius_m)
    speed_ms = 0.003
    movel([0.103618, -1.321882, -2.613498, -0.777009, 1.570796, 1.674414],accel_mss,speed_ms,0,blend_radius_m)
    speed_ms = 0.007
    movel([0.103637, -1.321609, -2.613669, -0.777111, 1.570796, 1.674433],accel_mss,speed_ms,0,blend_radius_m)
    movel([0.103885, -1.320476, -2.614373, -0.777540, 1.570796, 1.674681],accel_mss,speed_ms,0,blend_radius_m)
    movel([0.104417, -1.318992, -2.615294, -0.778103, 1.570796, 1.675214],accel_mss,speed_ms,0,blend_radius_m)
    movel([0.105039, -1.317574, -2.616171, -0.778644, 1.570796, 1.675836],accel_mss,speed_ms,0,blend_radius_m)
    movel([0.105483, -1.317048, -2.616496, -0.778845, 1.570796, 1.676279],accel_mss,speed_ms,0,blend_radius_m)
    movel([0.105791, -1.316870, -2.616606, -0.778914, 1.570796, 1.676587],accel_mss,speed_ms,0,blend_radius_m)
    movel([0.106222, -1.316711, -2.616703, -0.778974, 1.570796, 1.677018],accel_mss,speed_ms,0,blend_radius_m)
    movel([0.106665, -1.316600, -2.616772, -0.779017, 1.570796, 1.677462],accel_mss,speed_ms,0,blend_radius_m)
    movel([0.107028, -1.316570, -2.616790, -0.779028, 1.570796, 1.677825],accel_mss,speed_ms,0,blend_radius_m)
    movel([0.107242, -1.316675, -2.616726, -0.778988, 1.570796, 1.678039],accel_mss,speed_ms,0,blend_radius_m)
    movel([0.107306, -1.316943, -2.616561, -0.778886, 1.570796, 1.678102],accel_mss,speed_ms,0,blend_radius_m)
    movel([0.107218, -1.317538, -2.616193, -0.778658, 1.570796, 1.678014],accel_mss,speed_ms,0,blend_radius_m)
    movel([0.106840, -1.319216, -2.615155, -0.778018, 1.570796, 1.677636],accel_mss,speed_ms,0,blend_radius_m)
    movel([0.106420, -1.321002, -2.614046, -0.777340, 1.570796, 1.677217],accel_mss,speed_ms,0,blend_radius_m)
    movel([0.106260, -1.321559, -2.613699, -0.777130, 1.570796, 1.677056],accel_mss,speed_ms,0,blend_radius_m)
    movel([0.106100, -1.321846, -2.613521, -0.777022, 1.570796, 1.676897],accel_mss,speed_ms,0,blend_radius_m)
    movel([0.105428, -1.322200, -2.613300, -0.776889, 1.570796, 1.676224],accel_mss,speed_ms,0,blend_radius_m)
    movel([0.104756, -1.322315, -2.613228, -0.776846, 1.570796, 1.675553],accel_mss,speed_ms,0,blend_radius_m)
    movel([0.104107, -1.322373, -2.613192, -0.776824, 1.570796, 1.674903],accel_mss,speed_ms,0,blend_radius_m)
    movel([0.103793, -1.322308, -2.613233, -0.776848, 1.570796, 1.674589],accel_mss,speed_ms,0,blend_radius_m)
    movel([0.103635, -1.322082, -2.613374, -0.776933, 1.570796, 1.674432],accel_mss,speed_ms,0,blend_radius_m)
    speed_ms = 0.003
    movel([0.103618, -1.308235, -2.607092, -0.797062, 1.570796, 1.674414],accel_mss,speed_ms,0,blend_radius_m)
    speed_ms = 1.000
    movel([0.103618, -1.282197, -2.593889, -0.836303, 1.570796, 1.674414],accel_mss,speed_ms,0,blend_radius_m)
    movel([0.103813, -1.270306, -2.600804, -0.841279, 1.570796, 1.674610],accel_mss,speed_ms,0,blend_radius_m)
    movel([0.103813, -1.296516, -2.614163, -0.801711, 1.570796, 1.674610],accel_mss,speed_ms,0,blend_radius_m)
    speed_ms = 0.003
    movel([0.103813, -1.306788, -2.619039, -0.786562, 1.570796, 1.674610],accel_mss,speed_ms,0,blend_radius_m)
    speed_ms = 0.007
    movel([0.103818, -1.306456, -2.619240, -0.786693, 1.570796, 1.674615],accel_mss,speed_ms,0,blend_radius_m)
    movel([0.104142, -1.305715, -2.619687, -0.786987, 1.570796, 1.674938],accel_mss,speed_ms,0,blend_radius_m)
    movel([0.105377, -1.303033, -2.621301, -0.788055, 1.570796, 1.676173],accel_mss,speed_ms,0,blend_radius_m)
    movel([0.105952, -1.301774, -2.622055, -0.788560, 1.570796, 1.676748],accel_mss,speed_ms,0,blend_radius_m)
    movel([0.106444, -1.300670, -2.622715, -0.789004, 1.570796, 1.677240],accel_mss,speed_ms,0,blend_radius_m)
    movel([0.106854, -1.299726, -2.623277, -0.789385, 1.570796, 1.677650],accel_mss,speed_ms,0,blend_radius_m)
    movel([0.106834, -1.299363, -2.623494, -0.789532, 1.570796, 1.677630],accel_mss,speed_ms,0,blend_radius_m)
    movel([0.106601, -1.299322, -2.623518, -0.789549, 1.570796, 1.677397],accel_mss,speed_ms,0,blend_radius_m)
    movel([0.106084, -1.299434, -2.623451, -0.789504, 1.570796, 1.676881],accel_mss,speed_ms,0,blend_radius_m)
    movel([0.104894, -1.299801, -2.623233, -0.789355, 1.570796, 1.675691],accel_mss,speed_ms,0,blend_radius_m)
    movel([0.104141, -1.300033, -2.623094, -0.789261, 1.570796, 1.674938],accel_mss,speed_ms,0,blend_radius_m)
    movel([0.103630, -1.300168, -2.623014, -0.789207, 1.570796, 1.674427],accel_mss,speed_ms,0,blend_radius_m)
    movel([0.103281, -1.300238, -2.622973, -0.789179, 1.570796, 1.674077],accel_mss,speed_ms,0,blend_radius_m)
    movel([0.103139, -1.300064, -2.623076, -0.789249, 1.570796, 1.673936],accel_mss,speed_ms,0,blend_radius_m)
    movel([0.103501, -1.299189, -2.623597, -0.789603, 1.570796, 1.674298],accel_mss,speed_ms,0,blend_radius_m)
    movel([0.104030, -1.297983, -2.624314, -0.790092, 1.570796, 1.674826],accel_mss,speed_ms,0,blend_radius_m)
    movel([0.104855, -1.296189, -2.625376, -0.790824, 1.570796, 1.675651],accel_mss,speed_ms,0,blend_radius_m)
    movel([0.105571, -1.294665, -2.626275, -0.791449, 1.570796, 1.676367],accel_mss,speed_ms,0,blend_radius_m)
    movel([0.106206, -1.293339, -2.627055, -0.791995, 1.570796, 1.677002],accel_mss,speed_ms,0,blend_radius_m)
    movel([0.106762, -1.292196, -2.627726, -0.792467, 1.570796, 1.677558],accel_mss,speed_ms,0,blend_radius_m)
    movel([0.107086, -1.291849, -2.627929, -0.792611, 1.570796, 1.677883],accel_mss,speed_ms,0,blend_radius_m)
    movel([0.107542, -1.291653, -2.628044, -0.792692, 1.570796, 1.678339],accel_mss,speed_ms,0,blend_radius_m)
    movel([0.108293, -1.291386, -2.628200, -0.792803, 1.570796, 1.679089],accel_mss,speed_ms,0,blend_radius_m)
    movel([0.109705, -1.290927, -2.628468, -0.792993, 1.570796, 1.680502],accel_mss,speed_ms,0,blend_radius_m)
    movel([0.110994, -1.290524, -2.628704, -0.793161, 1.570796, 1.681790],accel_mss,speed_ms,0,blend_radius_m)
    movel([0.111769, -1.290303, -2.628832, -0.793253, 1.570796, 1.682565],accel_mss,speed_ms,0,blend_radius_m)
    movel([0.112276, -1.290181, -2.628904, -0.793304, 1.570796, 1.683072],accel_mss,speed_ms,0,blend_radius_m)
    movel([0.111888, -1.291179, -2.628321, -0.792889, 1.570796, 1.682685],accel_mss,speed_ms,0,blend_radius_m)
    movel([0.111324, -1.292151, -2.627752, -0.792486, 1.570796, 1.682120],accel_mss,speed_ms,0,blend_radius_m)
    movel([0.110646, -1.293277, -2.627092, -0.792020, 1.570796, 1.681442],accel_mss,speed_ms,0,blend_radius_m)
    movel([0.109696, -1.294842, -2.626171, -0.791376, 1.570796, 1.680492],accel_mss,speed_ms,0,blend_radius_m)
    movel([0.109237, -1.295653, -2.625692, -0.791043, 1.570796, 1.680034],accel_mss,speed_ms,0,blend_radius_m)
    movel([0.109006, -1.296136, -2.625407, -0.790845, 1.570796, 1.679802],accel_mss,speed_ms,0,blend_radius_m)
    movel([0.109167, -1.296352, -2.625280, -0.790757, 1.570796, 1.679964],accel_mss,speed_ms,0,blend_radius_m)
    movel([0.109462, -1.296309, -2.625305, -0.790775, 1.570796, 1.680258],accel_mss,speed_ms,0,blend_radius_m)
    movel([0.109933, -1.296190, -2.625375, -0.790823, 1.570796, 1.680729],accel_mss,speed_ms,0,blend_radius_m)
    movel([0.110719, -1.295949, -2.625518, -0.790922, 1.570796, 1.681516],accel_mss,speed_ms,0,blend_radius_m)
    movel([0.111646, -1.295667, -2.625685, -0.791038, 1.570796, 1.682443],accel_mss,speed_ms,0,blend_radius_m)
    movel([0.112117, -1.295551, -2.625753, -0.791085, 1.570796, 1.682914],accel_mss,speed_ms,0,blend_radius_m)
    movel([0.112419, -1.295641, -2.625700, -0.791048, 1.570796, 1.683215],accel_mss,speed_ms,0,blend_radius_m)
    movel([0.111167, -1.297314, -2.624710, -0.790364, 1.570796, 1.681963],accel_mss,speed_ms,0,blend_radius_m)
    movel([0.109797, -1.299108, -2.623645, -0.789635, 1.570796, 1.680593],accel_mss,speed_ms,0,blend_radius_m)
    movel([0.108182, -1.301220, -2.622386, -0.788783, 1.570796, 1.678978],accel_mss,speed_ms,0,blend_radius_m)
    movel([0.106560, -1.303325, -2.621126, -0.787938, 1.570796, 1.677356],accel_mss,speed_ms,0,blend_radius_m)
    movel([0.105169, -1.305112, -2.620051, -0.787226, 1.570796, 1.675965],accel_mss,speed_ms,0,blend_radius_m)
    movel([0.103939, -1.306679, -2.619105, -0.786605, 1.570796, 1.674736],accel_mss,speed_ms,0,blend_radius_m)
    speed_ms = 0.003
    movel([0.103813, -1.310267, -2.620648, -0.781474, 1.570796, 1.674610],accel_mss,speed_ms,0,blend_radius_m)
    speed_ms = 0.007
    movel([0.103818, -1.309935, -2.620849, -0.781604, 1.570796, 1.674615],accel_mss,speed_ms,0,blend_radius_m)
    movel([0.104142, -1.309196, -2.621298, -0.781895, 1.570796, 1.674938],accel_mss,speed_ms,0,blend_radius_m)
    movel([0.105377, -1.306521, -2.622916, -0.782952, 1.570796, 1.676173],accel_mss,speed_ms,0,blend_radius_m)
    movel([0.105952, -1.305264, -2.623673, -0.783452, 1.570796, 1.676748],accel_mss,speed_ms,0,blend_radius_m)
    movel([0.106444, -1.304162, -2.624334, -0.783892, 1.570796, 1.677240],accel_mss,speed_ms,0,blend_radius_m)
    movel([0.106854, -1.303221, -2.624898, -0.784270, 1.570796, 1.677650],accel_mss,speed_ms,0,blend_radius_m)
    movel([0.106834, -1.302859, -2.625115, -0.784415, 1.570796, 1.677630],accel_mss,speed_ms,0,blend_radius_m)
    movel([0.106601, -1.302818, -2.625140, -0.784432, 1.570796, 1.677397],accel_mss,speed_ms,0,blend_radius_m)
    movel([0.106084, -1.302929, -2.625073, -0.784387, 1.570796, 1.676881],accel_mss,speed_ms,0,blend_radius_m)
    movel([0.104894, -1.303295, -2.624854, -0.784240, 1.570796, 1.675691],accel_mss,speed_ms,0,blend_radius_m)
    movel([0.104141, -1.303528, -2.624715, -0.784147, 1.570796, 1.674938],accel_mss,speed_ms,0,blend_radius_m)
    movel([0.103630, -1.303662, -2.624634, -0.784093, 1.570796, 1.674427],accel_mss,speed_ms,0,blend_radius_m)
    movel([0.103281, -1.303731, -2.624593, -0.784065, 1.570796, 1.674077],accel_mss,speed_ms,0,blend_radius_m)
    movel([0.103139, -1.303558, -2.624696, -0.784134, 1.570796, 1.673936],accel_mss,speed_ms,0,blend_radius_m)
    movel([0.103501, -1.302685, -2.625219, -0.784485, 1.570796, 1.674298],accel_mss,speed_ms,0,blend_radius_m)
    movel([0.104030, -1.301482, -2.625938, -0.784970, 1.570796, 1.674826],accel_mss,speed_ms,0,blend_radius_m)
    movel([0.104855, -1.299692, -2.627003, -0.785694, 1.570796, 1.675651],accel_mss,speed_ms,0,blend_radius_m)
    movel([0.105571, -1.298171, -2.627905, -0.786313, 1.570796, 1.676367],accel_mss,speed_ms,0,blend_radius_m)
    movel([0.106206, -1.296848, -2.628687, -0.786854, 1.570796, 1.677002],accel_mss,speed_ms,0,blend_radius_m)
    movel([0.106762, -1.295708, -2.629359, -0.787322, 1.570796, 1.677558],accel_mss,speed_ms,0,blend_radius_m)
    movel([0.107086, -1.295361, -2.629563, -0.787464, 1.570796, 1.677883],accel_mss,speed_ms,0,blend_radius_m)
    movel([0.107542, -1.295166, -2.629678, -0.787545, 1.570796, 1.678339],accel_mss,speed_ms,0,blend_radius_m)
    movel([0.108293, -1.294899, -2.629835, -0.787655, 1.570796, 1.679089],accel_mss,speed_ms,0,blend_radius_m)
    movel([0.109705, -1.294442, -2.630104, -0.787843, 1.570796, 1.680502],accel_mss,speed_ms,0,blend_radius_m)
    movel([0.110994, -1.294039, -2.630340, -0.788010, 1.570796, 1.681790],accel_mss,speed_ms,0,blend_radius_m)
    movel([0.111769, -1.293819, -2.630469, -0.788101, 1.570796, 1.682565],accel_mss,speed_ms,0,blend_radius_m)
    movel([0.112276, -1.293697, -2.630541, -0.788151, 1.570796, 1.683072],accel_mss,speed_ms,0,blend_radius_m)
    movel([0.111888, -1.294693, -2.629956, -0.787740, 1.570796, 1.682685],accel_mss,speed_ms,0,blend_radius_m)
    movel([0.111324, -1.295663, -2.629386, -0.787340, 1.570796, 1.682120],accel_mss,speed_ms,0,blend_radius_m)
    movel([0.110646, -1.296786, -2.628724, -0.786879, 1.570796, 1.681442],accel_mss,speed_ms,0,blend_radius_m)
    movel([0.109696, -1.298348, -2.627800, -0.786241, 1.570796, 1.680492],accel_mss,speed_ms,0,blend_radius_m)
    movel([0.109237, -1.299157, -2.627320, -0.785911, 1.570796, 1.680034],accel_mss,speed_ms,0,blend_radius_m)
    movel([0.109006, -1.299639, -2.627034, -0.785716, 1.570796, 1.679802],accel_mss,speed_ms,0,blend_radius_m)
    movel([0.109167, -1.299855, -2.626906, -0.785628, 1.570796, 1.679964],accel_mss,speed_ms,0,blend_radius_m)
    movel([0.109462, -1.299811, -2.626932, -0.785646, 1.570796, 1.680258],accel_mss,speed_ms,0,blend_radius_m)
    movel([0.109933, -1.299693, -2.627002, -0.785694, 1.570796, 1.680729],accel_mss,speed_ms,0,blend_radius_m)
    movel([0.110719, -1.299452, -2.627145, -0.785791, 1.570796, 1.681516],accel_mss,speed_ms,0,blend_radius_m)
    movel([0.111646, -1.299170, -2.627312, -0.785906, 1.570796, 1.682443],accel_mss,speed_ms,0,blend_radius_m)
    movel([0.112117, -1.299056, -2.627381, -0.785953, 1.570796, 1.682914],accel_mss,speed_ms,0,blend_radius_m)
    movel([0.112419, -1.299145, -2.627327, -0.785916, 1.570796, 1.683215],accel_mss,speed_ms,0,blend_radius_m)
    movel([0.111167, -1.300815, -2.626335, -0.785239, 1.570796, 1.681963],accel_mss,speed_ms,0,blend_radius_m)
    movel([0.109797, -1.302605, -2.625267, -0.784517, 1.570796, 1.680593],accel_mss,speed_ms,0,blend_radius_m)
    movel([0.108182, -1.304712, -2.624004, -0.783673, 1.570796, 1.678978],accel_mss,speed_ms,0,blend_radius_m)
    movel([0.106560, -1.306812, -2.622741, -0.782837, 1.570796, 1.677356],accel_mss,speed_ms,0,blend_radius_m)
    movel([0.105169, -1.308594, -2.621663, -0.782132, 1.570796, 1.675965],accel_mss,speed_ms,0,blend_radius_m)
    movel([0.103939, -1.310158, -2.620714, -0.781517, 1.570796, 1.674736],accel_mss,speed_ms,0,blend_radius_m)
    speed_ms = 0.003
    movel([0.103813, -1.296516, -2.614163, -0.801711, 1.570796, 1.674610],accel_mss,speed_ms,0,blend_radius_m)
    speed_ms = 1.000
    movel([0.103813, -1.270306, -2.600804, -0.841279, 1.570796, 1.674610],accel_mss,speed_ms,0,blend_radius_m)
    movel([0.097054, -1.268961, -2.601575, -0.841853, 1.570796, 1.667851],accel_mss,speed_ms,0,blend_radius_m)
    movel([0.097054, -1.295189, -2.614952, -0.802248, 1.570796, 1.667851],accel_mss,speed_ms,0,blend_radius_m)
    speed_ms = 0.003
    movel([0.097054, -1.305471, -2.619835, -0.787084, 1.570796, 1.667851],accel_mss,speed_ms,0,blend_radius_m)
    speed_ms = 0.007
    movel([0.096828, -1.305732, -2.619677, -0.786980, 1.570796, 1.667624],accel_mss,speed_ms,0,blend_radius_m)
    movel([0.096502, -1.305914, -2.619567, -0.786908, 1.570796, 1.667298],accel_mss,speed_ms,0,blend_radius_m)
    movel([0.095838, -1.306121, -2.619442, -0.786826, 1.570796, 1.666635],accel_mss,speed_ms,0,blend_radius_m)
    movel([0.093053, -1.306885, -2.618981, -0.786524, 1.570796, 1.663849],accel_mss,speed_ms,0,blend_radius_m)
    movel([0.089387, -1.307997, -2.618307, -0.786085, 1.570796, 1.660183],accel_mss,speed_ms,0,blend_radius_m)
    movel([0.085759, -1.309319, -2.617504, -0.785565, 1.570796, 1.656556],accel_mss,speed_ms,0,blend_radius_m)
    movel([0.082322, -1.310790, -2.616608, -0.784990, 1.570796, 1.653118],accel_mss,speed_ms,0,blend_radius_m)
    movel([0.079223, -1.312346, -2.615658, -0.784385, 1.570796, 1.650019],accel_mss,speed_ms,0,blend_radius_m)
    movel([0.076467, -1.313922, -2.614692, -0.783776, 1.570796, 1.647263],accel_mss,speed_ms,0,blend_radius_m)
    movel([0.073248, -1.315908, -2.613469, -0.783012, 1.570796, 1.644045],accel_mss,speed_ms,0,blend_radius_m)
    movel([0.070195, -1.317895, -2.612241, -0.782253, 1.570796, 1.640991],accel_mss,speed_ms,0,blend_radius_m)
    movel([0.068013, -1.319445, -2.611279, -0.781664, 1.570796, 1.638809],accel_mss,speed_ms,0,blend_radius_m)
    movel([0.067576, -1.319730, -2.611102, -0.781557, 1.570796, 1.638372],accel_mss,speed_ms,0,blend_radius_m)
    movel([0.067261, -1.319825, -2.611043, -0.781521, 1.570796, 1.638057],accel_mss,speed_ms,0,blend_radius_m)
    movel([0.066994, -1.319754, -2.611087, -0.781548, 1.570796, 1.637790],accel_mss,speed_ms,0,blend_radius_m)
    movel([0.066710, -1.319488, -2.611253, -0.781648, 1.570796, 1.637506],accel_mss,speed_ms,0,blend_radius_m)
    movel([0.066534, -1.319145, -2.611466, -0.781778, 1.570796, 1.637330],accel_mss,speed_ms,0,blend_radius_m)
    movel([0.066526, -1.318728, -2.611725, -0.781936, 1.570796, 1.637323],accel_mss,speed_ms,0,blend_radius_m)
    movel([0.066594, -1.318467, -2.611886, -0.782035, 1.570796, 1.637390],accel_mss,speed_ms,0,blend_radius_m)
    movel([0.066867, -1.318064, -2.612136, -0.782189, 1.570796, 1.637663],accel_mss,speed_ms,0,blend_radius_m)
    movel([0.067167, -1.317788, -2.612307, -0.782293, 1.570796, 1.637963],accel_mss,speed_ms,0,blend_radius_m)
    movel([0.067720, -1.317344, -2.612582, -0.782463, 1.570796, 1.638516],accel_mss,speed_ms,0,blend_radius_m)
    movel([0.068900, -1.316468, -2.613124, -0.782797, 1.570796, 1.639696],accel_mss,speed_ms,0,blend_radius_m)
    movel([0.070231, -1.315498, -2.613722, -0.783169, 1.570796, 1.641027],accel_mss,speed_ms,0,blend_radius_m)
    movel([0.071504, -1.314595, -2.614278, -0.783516, 1.570796, 1.642300],accel_mss,speed_ms,0,blend_radius_m)
    movel([0.073287, -1.313443, -2.614985, -0.783960, 1.570796, 1.644084],accel_mss,speed_ms,0,blend_radius_m)
    movel([0.076248, -1.311728, -2.616036, -0.784625, 1.570796, 1.647044],accel_mss,speed_ms,0,blend_radius_m)
    movel([0.079336, -1.310023, -2.617076, -0.785290, 1.570796, 1.650133],accel_mss,speed_ms,0,blend_radius_m)
    movel([0.081717, -1.308817, -2.617810, -0.785763, 1.570796, 1.652514],accel_mss,speed_ms,0,blend_radius_m)
    movel([0.083889, -1.307824, -2.618412, -0.786153, 1.570796, 1.654686],accel_mss,speed_ms,0,blend_radius_m)
    movel([0.085940, -1.306966, -2.618932, -0.786491, 1.570796, 1.656736],accel_mss,speed_ms,0,blend_radius_m)
    movel([0.088113, -1.306152, -2.619424, -0.786813, 1.570796, 1.658909],accel_mss,speed_ms,0,blend_radius_m)
    movel([0.090652, -1.305288, -2.619945, -0.787156, 1.570796, 1.661449],accel_mss,speed_ms,0,blend_radius_m)
    movel([0.093223, -1.304484, -2.620429, -0.787476, 1.570796, 1.664019],accel_mss,speed_ms,0,blend_radius_m)
    movel([0.095145, -1.303969, -2.620739, -0.787681, 1.570796, 1.665941],accel_mss,speed_ms,0,blend_radius_m)
    movel([0.096536, -1.303696, -2.620903, -0.787790, 1.570796, 1.667333],accel_mss,speed_ms,0,blend_radius_m)
    movel([0.097274, -1.303722, -2.620887, -0.787780, 1.570796, 1.668070],accel_mss,speed_ms,0,blend_radius_m)
    movel([0.097500, -1.303897, -2.620782, -0.787710, 1.570796, 1.668297],accel_mss,speed_ms,0,blend_radius_m)
    movel([0.097411, -1.304460, -2.620444, -0.787485, 1.570796, 1.668208],accel_mss,speed_ms,0,blend_radius_m)
    movel([0.097336, -1.304739, -2.620276, -0.787374, 1.570796, 1.668132],accel_mss,speed_ms,0,blend_radius_m)
    movel([0.097240, -1.305028, -2.620101, -0.787259, 1.570796, 1.668037],accel_mss,speed_ms,0,blend_radius_m)
    movel([0.097140, -1.305291, -2.619943, -0.787155, 1.570796, 1.667936],accel_mss,speed_ms,0,blend_radius_m)
    speed_ms = 0.003
    movel([0.097054, -1.308952, -2.621446, -0.781991, 1.570796, 1.667851],accel_mss,speed_ms,0,blend_radius_m)
    speed_ms = 0.007
    movel([0.096828, -1.309213, -2.621288, -0.781888, 1.570796, 1.667624],accel_mss,speed_ms,0,blend_radius_m)
    movel([0.096502, -1.309395, -2.621178, -0.781817, 1.570796, 1.667298],accel_mss,speed_ms,0,blend_radius_m)
    movel([0.095838, -1.309601, -2.621052, -0.781735, 1.570796, 1.666635],accel_mss,speed_ms,0,blend_radius_m)
    movel([0.093053, -1.310363, -2.620589, -0.781436, 1.570796, 1.663849],accel_mss,speed_ms,0,blend_radius_m)
    movel([0.089387, -1.311473, -2.619914, -0.781002, 1.570796, 1.660183],accel_mss,speed_ms,0,blend_radius_m)
    movel([0.085759, -1.312792, -2.619109, -0.780488, 1.570796, 1.656556],accel_mss,speed_ms,0,blend_radius_m)
    movel([0.082322, -1.314260, -2.618210, -0.779919, 1.570796, 1.653118],accel_mss,speed_ms,0,blend_radius_m)
    movel([0.079223, -1.315812, -2.617257, -0.779320, 1.570796, 1.650019],accel_mss,speed_ms,0,blend_radius_m)
    movel([0.076467, -1.317384, -2.616288, -0.778717, 1.570796, 1.647263],accel_mss,speed_ms,0,blend_radius_m)
    movel([0.073248, -1.319365, -2.615063, -0.777961, 1.570796, 1.644045],accel_mss,speed_ms,0,blend_radius_m)
    movel([0.070195, -1.321348, -2.613831, -0.777210, 1.570796, 1.640991],accel_mss,speed_ms,0,blend_radius_m)
    movel([0.068013, -1.322894, -2.612867, -0.776628, 1.570796, 1.638809],accel_mss,speed_ms,0,blend_radius_m)
    movel([0.067576, -1.323178, -2.612689, -0.776521, 1.570796, 1.638372],accel_mss,speed_ms,0,blend_radius_m)
    movel([0.067261, -1.323273, -2.612630, -0.776486, 1.570796, 1.638057],accel_mss,speed_ms,0,blend_radius_m)
    movel([0.066994, -1.323202, -2.612674, -0.776512, 1.570796, 1.637790],accel_mss,speed_ms,0,blend_radius_m)
    movel([0.066710, -1.322937, -2.612840, -0.776612, 1.570796, 1.637506],accel_mss,speed_ms,0,blend_radius_m)
    movel([0.066534, -1.322594, -2.613054, -0.776741, 1.570796, 1.637330],accel_mss,speed_ms,0,blend_radius_m)
    movel([0.066526, -1.322178, -2.613314, -0.776897, 1.570796, 1.637323],accel_mss,speed_ms,0,blend_radius_m)
    movel([0.066594, -1.321919, -2.613475, -0.776995, 1.570796, 1.637390],accel_mss,speed_ms,0,blend_radius_m)
    movel([0.066867, -1.321516, -2.613726, -0.777146, 1.570796, 1.637663],accel_mss,speed_ms,0,blend_radius_m)
    movel([0.067167, -1.321241, -2.613897, -0.777250, 1.570796, 1.637963],accel_mss,speed_ms,0,blend_radius_m)
    movel([0.067720, -1.320799, -2.614173, -0.777418, 1.570796, 1.638516],accel_mss,speed_ms,0,blend_radius_m)
    movel([0.068900, -1.319924, -2.614716, -0.777749, 1.570796, 1.639696],accel_mss,speed_ms,0,blend_radius_m)
    movel([0.070231, -1.318957, -2.615316, -0.778116, 1.570796, 1.641027],accel_mss,speed_ms,0,blend_radius_m)
    movel([0.071504, -1.318055, -2.615874, -0.778460, 1.570796, 1.642300],accel_mss,speed_ms,0,blend_radius_m)
    movel([0.073287, -1.316906, -2.616583, -0.778900, 1.570796, 1.644084],accel_mss,speed_ms,0,blend_radius_m)
    movel([0.076248, -1.315195, -2.617636, -0.779558, 1.570796, 1.647044],accel_mss,speed_ms,0,blend_radius_m)
    movel([0.079336, -1.313494, -2.618679, -0.780215, 1.570796, 1.650133],accel_mss,speed_ms,0,blend_radius_m)
    movel([0.081717, -1.312291, -2.619415, -0.780683, 1.570796, 1.652514],accel_mss,speed_ms,0,blend_radius_m)
    movel([0.083889, -1.311300, -2.620019, -0.781070, 1.570796, 1.654686],accel_mss,speed_ms,0,blend_radius_m)
    movel([0.085940, -1.310444, -2.620540, -0.781405, 1.570796, 1.656736],accel_mss,speed_ms,0,blend_radius_m)
    movel([0.088113, -1.309632, -2.621034, -0.781723, 1.570796, 1.658909],accel_mss,speed_ms,0,blend_radius_m)
    movel([0.090652, -1.308770, -2.621556, -0.782062, 1.570796, 1.661449],accel_mss,speed_ms,0,blend_radius_m)
    movel([0.093223, -1.307968, -2.622042, -0.782379, 1.570796, 1.664019],accel_mss,speed_ms,0,blend_radius_m)
    movel([0.095145, -1.307454, -2.622353, -0.782582, 1.570796, 1.665941],accel_mss,speed_ms,0,blend_radius_m)
    movel([0.096536, -1.307182, -2.622517, -0.782690, 1.570796, 1.667333],accel_mss,speed_ms,0,blend_radius_m)
    movel([0.097274, -1.307208, -2.622501, -0.782680, 1.570796, 1.668070],accel_mss,speed_ms,0,blend_radius_m)
    movel([0.097500, -1.307382, -2.622396, -0.782611, 1.570796, 1.668297],accel_mss,speed_ms,0,blend_radius_m)
    movel([0.097411, -1.307944, -2.622056, -0.782389, 1.570796, 1.668208],accel_mss,speed_ms,0,blend_radius_m)
    movel([0.097336, -1.308222, -2.621888, -0.782279, 1.570796, 1.668132],accel_mss,speed_ms,0,blend_radius_m)
    movel([0.097240, -1.308511, -2.621713, -0.782165, 1.570796, 1.668037],accel_mss,speed_ms,0,blend_radius_m)
    movel([0.097140, -1.308774, -2.621554, -0.782061, 1.570796, 1.667936],accel_mss,speed_ms,0,blend_radius_m)
    speed_ms = 0.003
    movel([0.097054, -1.295189, -2.614952, -0.802248, 1.570796, 1.667851],accel_mss,speed_ms,0,blend_radius_m)
    speed_ms = 1.000
    movel([0.097054, -1.268961, -2.601575, -0.841853, 1.570796, 1.667851],accel_mss,speed_ms,0,blend_radius_m)
    movel([0.095455, -1.266877, -2.602766, -0.842746, 1.570796, 1.666251],accel_mss,speed_ms,0,blend_radius_m)
    movel([0.095455, -1.293135, -2.616170, -0.803084, 1.570796, 1.666251],accel_mss,speed_ms,0,blend_radius_m)
    speed_ms = 0.003
    movel([0.095455, -1.303429, -2.621063, -0.787897, 1.570796, 1.666251],accel_mss,speed_ms,0,blend_radius_m)
    speed_ms = 0.007
    movel([0.094815, -1.303693, -2.620905, -0.787791, 1.570796, 1.665611],accel_mss,speed_ms,0,blend_radius_m)
    movel([0.093768, -1.303954, -2.620748, -0.787687, 1.570796, 1.664565],accel_mss,speed_ms,0,blend_radius_m)
    movel([0.093133, -1.304102, -2.620659, -0.787628, 1.570796, 1.663930],accel_mss,speed_ms,0,blend_radius_m)
    movel([0.092577, -1.304211, -2.620593, -0.787584, 1.570796, 1.663373],accel_mss,speed_ms,0,blend_radius_m)
    movel([0.092119, -1.304286, -2.620548, -0.787555, 1.570796, 1.662915],accel_mss,speed_ms,0,blend_radius_m)
    movel([0.091857, -1.304106, -2.620657, -0.787627, 1.570796, 1.662654],accel_mss,speed_ms,0,blend_radius_m)
    movel([0.091804, -1.303854, -2.620808, -0.787727, 1.570796, 1.662600],accel_mss,speed_ms,0,blend_radius_m)
    movel([0.091848, -1.303588, -2.620968, -0.787833, 1.570796, 1.662644],accel_mss,speed_ms,0,blend_radius_m)
    movel([0.092415, -1.303110, -2.621254, -0.788024, 1.570796, 1.663211],accel_mss,speed_ms,0,blend_radius_m)
    movel([0.093796, -1.302701, -2.621500, -0.788188, 1.570796, 1.664592],accel_mss,speed_ms,0,blend_radius_m)
    movel([0.095147, -1.302357, -2.621706, -0.788326, 1.570796, 1.665943],accel_mss,speed_ms,0,blend_radius_m)
    movel([0.095680, -1.302353, -2.621709, -0.788328, 1.570796, 1.666476],accel_mss,speed_ms,0,blend_radius_m)
    movel([0.095880, -1.302466, -2.621641, -0.788282, 1.570796, 1.666676],accel_mss,speed_ms,0,blend_radius_m)
    movel([0.095874, -1.302908, -2.621376, -0.788105, 1.570796, 1.666670],accel_mss,speed_ms,0,blend_radius_m)
    movel([0.095665, -1.303223, -2.621187, -0.787979, 1.570796, 1.666461],accel_mss,speed_ms,0,blend_radius_m)
    speed_ms = 0.003
    movel([0.095455, -1.306916, -2.622678, -0.782796, 1.570796, 1.666251],accel_mss,speed_ms,0,blend_radius_m)
    speed_ms = 0.007
    movel([0.094815, -1.307179, -2.622519, -0.782691, 1.570796, 1.665611],accel_mss,speed_ms,0,blend_radius_m)
    movel([0.093768, -1.307439, -2.622362, -0.782588, 1.570796, 1.664565],accel_mss,speed_ms,0,blend_radius_m)
    movel([0.093133, -1.307587, -2.622272, -0.782530, 1.570796, 1.663930],accel_mss,speed_ms,0,blend_radius_m)
    movel([0.092577, -1.307696, -2.622206, -0.782487, 1.570796, 1.663373],accel_mss,speed_ms,0,blend_radius_m)
    movel([0.092119, -1.307771, -2.622161, -0.782457, 1.570796, 1.662915],accel_mss,speed_ms,0,blend_radius_m)
    movel([0.091857, -1.307590, -2.622270, -0.782528, 1.570796, 1.662654],accel_mss,speed_ms,0,blend_radius_m)
    movel([0.091804, -1.307340, -2.622422, -0.782628, 1.570796, 1.662600],accel_mss,speed_ms,0,blend_radius_m)
    movel([0.091848, -1.307074, -2.622582, -0.782733, 1.570796, 1.662644],accel_mss,speed_ms,0,blend_radius_m)
    movel([0.092415, -1.306598, -2.622870, -0.782922, 1.570796, 1.663211],accel_mss,speed_ms,0,blend_radius_m)
    movel([0.093796, -1.306189, -2.623116, -0.783084, 1.570796, 1.664592],accel_mss,speed_ms,0,blend_radius_m)
    movel([0.095147, -1.305846, -2.623322, -0.783220, 1.570796, 1.665943],accel_mss,speed_ms,0,blend_radius_m)
    movel([0.095680, -1.305842, -2.623325, -0.783222, 1.570796, 1.666476],accel_mss,speed_ms,0,blend_radius_m)
    movel([0.095880, -1.305954, -2.623257, -0.783177, 1.570796, 1.666676],accel_mss,speed_ms,0,blend_radius_m)
    movel([0.095874, -1.306395, -2.622992, -0.783002, 1.570796, 1.666670],accel_mss,speed_ms,0,blend_radius_m)
    movel([0.095665, -1.306710, -2.622802, -0.782877, 1.570796, 1.666461],accel_mss,speed_ms,0,blend_radius_m)
    speed_ms = 0.003
    movel([0.095455, -1.293135, -2.616170, -0.803084, 1.570796, 1.666251],accel_mss,speed_ms,0,blend_radius_m)
    speed_ms = 1.000
    movel([0.095455, -1.266877, -2.602766, -0.842746, 1.570796, 1.666251],accel_mss,speed_ms,0,blend_radius_m)
    movel([0.095405, -1.265298, -2.603664, -0.843426, 1.570796, 1.666201],accel_mss,speed_ms,0,blend_radius_m)
    movel([0.095405, -1.291578, -2.617089, -0.803722, 1.570796, 1.666201],accel_mss,speed_ms,0,blend_radius_m)
    speed_ms = 0.003
    movel([0.095405, -1.301882, -2.621990, -0.788516, 1.570796, 1.666201],accel_mss,speed_ms,0,blend_radius_m)
    speed_ms = 0.007
    movel([0.093973, -1.302304, -2.621738, -0.788347, 1.570796, 1.664770],accel_mss,speed_ms,0,blend_radius_m)
    movel([0.092537, -1.302698, -2.621502, -0.788189, 1.570796, 1.663334],accel_mss,speed_ms,0,blend_radius_m)
    movel([0.092269, -1.302658, -2.621526, -0.788205, 1.570796, 1.663065],accel_mss,speed_ms,0,blend_radius_m)
    movel([0.092184, -1.302449, -2.621651, -0.788289, 1.570796, 1.662981],accel_mss,speed_ms,0,blend_radius_m)
    movel([0.092128, -1.302079, -2.621873, -0.788437, 1.570796, 1.662924],accel_mss,speed_ms,0,blend_radius_m)
    movel([0.092124, -1.301814, -2.622031, -0.788544, 1.570796, 1.662920],accel_mss,speed_ms,0,blend_radius_m)
    movel([0.092244, -1.301453, -2.622247, -0.788689, 1.570796, 1.663040],accel_mss,speed_ms,0,blend_radius_m)
    movel([0.093053, -1.300803, -2.622635, -0.788951, 1.570796, 1.663849],accel_mss,speed_ms,0,blend_radius_m)
    movel([0.094199, -1.300463, -2.622838, -0.789088, 1.570796, 1.664996],accel_mss,speed_ms,0,blend_radius_m)
    movel([0.095309, -1.300319, -2.622924, -0.789146, 1.570796, 1.666105],accel_mss,speed_ms,0,blend_radius_m)
    movel([0.095864, -1.300514, -2.622808, -0.789067, 1.570796, 1.666660],accel_mss,speed_ms,0,blend_radius_m)
    movel([0.095977, -1.300744, -2.622670, -0.788974, 1.570796, 1.666773],accel_mss,speed_ms,0,blend_radius_m)
    movel([0.095993, -1.301082, -2.622469, -0.788838, 1.570796, 1.666789],accel_mss,speed_ms,0,blend_radius_m)
    movel([0.095919, -1.301425, -2.622264, -0.788700, 1.570796, 1.666715],accel_mss,speed_ms,0,blend_radius_m)
    movel([0.095405, -1.301882, -2.621990, -0.788516, 1.570796, 1.666201],accel_mss,speed_ms,0,blend_radius_m)
    speed_ms = 0.003
    movel([0.095405, -1.305372, -2.623608, -0.783409, 1.570796, 1.666201],accel_mss,speed_ms,0,blend_radius_m)
    speed_ms = 0.007
    movel([0.093973, -1.305793, -2.623354, -0.783242, 1.570796, 1.664770],accel_mss,speed_ms,0,blend_radius_m)
    movel([0.092537, -1.306187, -2.623117, -0.783085, 1.570796, 1.663334],accel_mss,speed_ms,0,blend_radius_m)
    movel([0.092269, -1.306146, -2.623142, -0.783101, 1.570796, 1.663065],accel_mss,speed_ms,0,blend_radius_m)
    movel([0.092184, -1.305938, -2.623267, -0.783184, 1.570796, 1.662981],accel_mss,speed_ms,0,blend_radius_m)
    movel([0.092128, -1.305569, -2.623489, -0.783331, 1.570796, 1.662924],accel_mss,speed_ms,0,blend_radius_m)
    movel([0.092124, -1.305304, -2.623649, -0.783437, 1.570796, 1.662920],accel_mss,speed_ms,0,blend_radius_m)
    movel([0.092244, -1.304944, -2.623865, -0.783580, 1.570796, 1.663040],accel_mss,speed_ms,0,blend_radius_m)
    movel([0.093053, -1.304296, -2.624254, -0.783839, 1.570796, 1.663849],accel_mss,speed_ms,0,blend_radius_m)
    movel([0.094199, -1.303956, -2.624458, -0.783975, 1.570796, 1.664996],accel_mss,speed_ms,0,blend_radius_m)
    movel([0.095309, -1.303812, -2.624544, -0.784033, 1.570796, 1.666105],accel_mss,speed_ms,0,blend_radius_m)
    movel([0.095864, -1.304007, -2.624428, -0.783955, 1.570796, 1.666660],accel_mss,speed_ms,0,blend_radius_m)
    movel([0.095977, -1.304237, -2.624289, -0.783863, 1.570796, 1.666773],accel_mss,speed_ms,0,blend_radius_m)
    movel([0.095993, -1.304573, -2.624088, -0.783728, 1.570796, 1.666789],accel_mss,speed_ms,0,blend_radius_m)
    movel([0.095919, -1.304916, -2.623882, -0.783591, 1.570796, 1.666715],accel_mss,speed_ms,0,blend_radius_m)
    movel([0.095405, -1.305372, -2.623608, -0.783409, 1.570796, 1.666201],accel_mss,speed_ms,0,blend_radius_m)
    speed_ms = 0.003
    movel([0.095405, -1.291578, -2.617089, -0.803722, 1.570796, 1.666201],accel_mss,speed_ms,0,blend_radius_m)
    speed_ms = 1.000
    movel([0.095405, -1.265298, -2.603664, -0.843426, 1.570796, 1.666201],accel_mss,speed_ms,0,blend_radius_m)
    movel([0.086620, -1.269064, -2.601516, -0.841809, 1.570796, 1.657416],accel_mss,speed_ms,0,blend_radius_m)
    movel([0.086620, -1.295291, -2.614891, -0.802207, 1.570796, 1.657416],accel_mss,speed_ms,0,blend_radius_m)
    speed_ms = 0.003
    movel([0.086620, -1.305571, -2.619774, -0.787044, 1.570796, 1.657416],accel_mss,speed_ms,0,blend_radius_m)
    speed_ms = 0.007
    movel([0.086582, -1.306010, -2.619509, -0.786870, 1.570796, 1.657378],accel_mss,speed_ms,0,blend_radius_m)
    movel([0.086379, -1.306296, -2.619337, -0.786757, 1.570796, 1.657175],accel_mss,speed_ms,0,blend_radius_m)
    movel([0.085833, -1.306567, -2.619173, -0.786649, 1.570796, 1.656630],accel_mss,speed_ms,0,blend_radius_m)
    movel([0.085166, -1.306876, -2.618986, -0.786527, 1.570796, 1.655962],accel_mss,speed_ms,0,blend_radius_m)
    movel([0.084376, -1.307221, -2.618777, -0.786391, 1.570796, 1.655172],accel_mss,speed_ms,0,blend_radius_m)
    movel([0.082276, -1.308128, -2.618228, -0.786033, 1.570796, 1.653073],accel_mss,speed_ms,0,blend_radius_m)
    movel([0.080804, -1.308806, -2.617816, -0.785767, 1.570796, 1.651600],accel_mss,speed_ms,0,blend_radius_m)
    movel([0.079595, -1.309416, -2.617445, -0.785528, 1.570796, 1.650391],accel_mss,speed_ms,0,blend_radius_m)
    movel([0.078387, -1.310089, -2.617036, -0.785264, 1.570796, 1.649183],accel_mss,speed_ms,0,blend_radius_m)
    movel([0.077797, -1.310425, -2.616831, -0.785133, 1.570796, 1.648593],accel_mss,speed_ms,0,blend_radius_m)
    movel([0.077272, -1.310708, -2.616659, -0.785023, 1.570796, 1.648069],accel_mss,speed_ms,0,blend_radius_m)
    movel([0.076832, -1.310931, -2.616522, -0.784935, 1.570796, 1.647629],accel_mss,speed_ms,0,blend_radius_m)
    movel([0.076556, -1.310865, -2.616563, -0.784961, 1.570796, 1.647352],accel_mss,speed_ms,0,blend_radius_m)
    movel([0.076460, -1.310625, -2.616709, -0.785055, 1.570796, 1.647257],accel_mss,speed_ms,0,blend_radius_m)
    movel([0.076484, -1.310298, -2.616908, -0.785183, 1.570796, 1.647280],accel_mss,speed_ms,0,blend_radius_m)
    movel([0.076654, -1.309989, -2.617097, -0.785303, 1.570796, 1.647450],accel_mss,speed_ms,0,blend_radius_m)
    movel([0.077020, -1.309644, -2.617307, -0.785438, 1.570796, 1.647816],accel_mss,speed_ms,0,blend_radius_m)
    movel([0.077663, -1.309194, -2.617580, -0.785615, 1.570796, 1.648459],accel_mss,speed_ms,0,blend_radius_m)
    movel([0.078607, -1.308648, -2.617912, -0.785829, 1.570796, 1.649403],accel_mss,speed_ms,0,blend_radius_m)
    movel([0.080873, -1.307513, -2.618601, -0.786276, 1.570796, 1.651669],accel_mss,speed_ms,0,blend_radius_m)
    movel([0.083162, -1.306405, -2.619271, -0.786713, 1.570796, 1.653958],accel_mss,speed_ms,0,blend_radius_m)
    movel([0.084650, -1.305747, -2.619668, -0.786974, 1.570796, 1.655447],accel_mss,speed_ms,0,blend_radius_m)
    movel([0.085312, -1.305509, -2.619812, -0.787068, 1.570796, 1.656108],accel_mss,speed_ms,0,blend_radius_m)
    movel([0.085892, -1.305370, -2.619896, -0.787124, 1.570796, 1.656689],accel_mss,speed_ms,0,blend_radius_m)
    movel([0.086338, -1.305334, -2.619917, -0.787138, 1.570796, 1.657135],accel_mss,speed_ms,0,blend_radius_m)
    movel([0.086557, -1.305429, -2.619860, -0.787100, 1.570796, 1.657353],accel_mss,speed_ms,0,blend_radius_m)
    speed_ms = 0.003
    movel([0.086620, -1.309053, -2.621385, -0.781951, 1.570796, 1.657416],accel_mss,speed_ms,0,blend_radius_m)
    speed_ms = 0.007
    movel([0.086582, -1.309490, -2.621120, -0.781779, 1.570796, 1.657378],accel_mss,speed_ms,0,blend_radius_m)
    movel([0.086379, -1.309776, -2.620947, -0.781667, 1.570796, 1.657175],accel_mss,speed_ms,0,blend_radius_m)
    movel([0.085833, -1.310046, -2.620782, -0.781561, 1.570796, 1.656630],accel_mss,speed_ms,0,blend_radius_m)
    movel([0.085166, -1.310354, -2.620595, -0.781440, 1.570796, 1.655962],accel_mss,speed_ms,0,blend_radius_m)
    movel([0.084376, -1.310699, -2.620385, -0.781305, 1.570796, 1.655172],accel_mss,speed_ms,0,blend_radius_m)
    movel([0.082276, -1.311603, -2.619834, -0.780951, 1.570796, 1.653073],accel_mss,speed_ms,0,blend_radius_m)
    movel([0.080804, -1.312280, -2.619421, -0.780687, 1.570796, 1.651600],accel_mss,speed_ms,0,blend_radius_m)
    movel([0.079595, -1.312889, -2.619050, -0.780450, 1.570796, 1.650391],accel_mss,speed_ms,0,blend_radius_m)
    movel([0.078387, -1.313560, -2.618639, -0.780190, 1.570796, 1.649183],accel_mss,speed_ms,0,blend_radius_m)
    movel([0.077797, -1.313896, -2.618434, -0.780060, 1.570796, 1.648593],accel_mss,speed_ms,0,blend_radius_m)
    movel([0.077272, -1.314177, -2.618261, -0.779951, 1.570796, 1.648069],accel_mss,speed_ms,0,blend_radius_m)
    movel([0.076832, -1.314401, -2.618124, -0.779864, 1.570796, 1.647629],accel_mss,speed_ms,0,blend_radius_m)
    movel([0.076556, -1.314335, -2.618165, -0.779890, 1.570796, 1.647352],accel_mss,speed_ms,0,blend_radius_m)
    movel([0.076460, -1.314095, -2.618312, -0.779983, 1.570796, 1.647257],accel_mss,speed_ms,0,blend_radius_m)
    movel([0.076484, -1.313769, -2.618511, -0.780109, 1.570796, 1.647280],accel_mss,speed_ms,0,blend_radius_m)
    movel([0.076654, -1.313460, -2.618700, -0.780229, 1.570796, 1.647450],accel_mss,speed_ms,0,blend_radius_m)
    movel([0.077020, -1.313116, -2.618911, -0.780362, 1.570796, 1.647816],accel_mss,speed_ms,0,blend_radius_m)
    movel([0.077663, -1.312667, -2.619185, -0.780537, 1.570796, 1.648459],accel_mss,speed_ms,0,blend_radius_m)
    movel([0.078607, -1.312122, -2.619518, -0.780749, 1.570796, 1.649403],accel_mss,speed_ms,0,blend_radius_m)
    movel([0.080873, -1.310990, -2.620208, -0.781191, 1.570796, 1.651669],accel_mss,speed_ms,0,blend_radius_m)
    movel([0.083162, -1.309885, -2.620880, -0.781624, 1.570796, 1.653958],accel_mss,speed_ms,0,blend_radius_m)
    movel([0.084650, -1.309228, -2.621279, -0.781882, 1.570796, 1.655447],accel_mss,speed_ms,0,blend_radius_m)
    movel([0.085312, -1.308990, -2.621423, -0.781976, 1.570796, 1.656108],accel_mss,speed_ms,0,blend_radius_m)
    movel([0.085892, -1.308852, -2.621507, -0.782030, 1.570796, 1.656689],accel_mss,speed_ms,0,blend_radius_m)
    movel([0.086338, -1.308816, -2.621529, -0.782044, 1.570796, 1.657135],accel_mss,speed_ms,0,blend_radius_m)
    movel([0.086557, -1.308911, -2.621471, -0.782007, 1.570796, 1.657353],accel_mss,speed_ms,0,blend_radius_m)
    speed_ms = 0.003
    movel([0.086620, -1.295291, -2.614891, -0.802207, 1.570796, 1.657416],accel_mss,speed_ms,0,blend_radius_m)
    speed_ms = 1.000
    movel([0.086620, -1.269064, -2.601516, -0.841809, 1.570796, 1.657416],accel_mss,speed_ms,0,blend_radius_m)
    movel([0.086236, -1.268202, -2.602010, -0.842178, 1.570796, 1.657033],accel_mss,speed_ms,0,blend_radius_m)
    movel([0.086236, -1.294441, -2.615396, -0.802552, 1.570796, 1.657033],accel_mss,speed_ms,0,blend_radius_m)
    speed_ms = 0.003
    movel([0.086236, -1.304727, -2.620283, -0.787379, 1.570796, 1.657033],accel_mss,speed_ms,0,blend_radius_m)
    speed_ms = 0.007
    movel([0.085836, -1.304918, -2.620168, -0.787303, 1.570796, 1.656632],accel_mss,speed_ms,0,blend_radius_m)
    movel([0.085399, -1.305046, -2.620090, -0.787252, 1.570796, 1.656196],accel_mss,speed_ms,0,blend_radius_m)
    movel([0.085110, -1.304940, -2.620155, -0.787294, 1.570796, 1.655906],accel_mss,speed_ms,0,blend_radius_m)
    movel([0.085056, -1.304704, -2.620297, -0.787388, 1.570796, 1.655852],accel_mss,speed_ms,0,blend_radius_m)
    movel([0.085010, -1.304411, -2.620473, -0.787505, 1.570796, 1.655807],accel_mss,speed_ms,0,blend_radius_m)
    movel([0.084978, -1.304084, -2.620670, -0.787635, 1.570796, 1.655775],accel_mss,speed_ms,0,blend_radius_m)
    movel([0.084892, -1.303468, -2.621040, -0.787881, 1.570796, 1.655688],accel_mss,speed_ms,0,blend_radius_m)
    movel([0.084735, -1.303084, -2.621270, -0.788035, 1.570796, 1.655531],accel_mss,speed_ms,0,blend_radius_m)
    movel([0.084474, -1.302865, -2.621402, -0.788122, 1.570796, 1.655271],accel_mss,speed_ms,0,blend_radius_m)
    movel([0.084085, -1.302763, -2.621463, -0.788163, 1.570796, 1.654882],accel_mss,speed_ms,0,blend_radius_m)
    movel([0.083756, -1.302782, -2.621451, -0.788155, 1.570796, 1.654553],accel_mss,speed_ms,0,blend_radius_m)
    movel([0.083385, -1.302888, -2.621388, -0.788113, 1.570796, 1.654181],accel_mss,speed_ms,0,blend_radius_m)
    movel([0.082789, -1.303141, -2.621236, -0.788012, 1.570796, 1.653585],accel_mss,speed_ms,0,blend_radius_m)
    movel([0.081437, -1.303782, -2.620851, -0.787756, 1.570796, 1.652233],accel_mss,speed_ms,0,blend_radius_m)
    movel([0.079639, -1.304655, -2.620326, -0.787408, 1.570796, 1.650435],accel_mss,speed_ms,0,blend_radius_m)
    movel([0.078834, -1.305092, -2.620063, -0.787234, 1.570796, 1.649630],accel_mss,speed_ms,0,blend_radius_m)
    movel([0.078346, -1.305441, -2.619853, -0.787095, 1.570796, 1.649142],accel_mss,speed_ms,0,blend_radius_m)
    movel([0.077948, -1.305852, -2.619605, -0.786932, 1.570796, 1.648744],accel_mss,speed_ms,0,blend_radius_m)
    movel([0.077690, -1.306269, -2.619353, -0.786767, 1.570796, 1.648486],accel_mss,speed_ms,0,blend_radius_m)
    movel([0.077544, -1.306721, -2.619080, -0.786588, 1.570796, 1.648340],accel_mss,speed_ms,0,blend_radius_m)
    movel([0.077508, -1.307216, -2.618780, -0.786393, 1.570796, 1.648304],accel_mss,speed_ms,0,blend_radius_m)
    movel([0.077587, -1.307758, -2.618452, -0.786179, 1.570796, 1.648383],accel_mss,speed_ms,0,blend_radius_m)
    movel([0.077671, -1.308128, -2.618228, -0.786033, 1.570796, 1.648467],accel_mss,speed_ms,0,blend_radius_m)
    movel([0.077735, -1.308415, -2.618054, -0.785921, 1.570796, 1.648531],accel_mss,speed_ms,0,blend_radius_m)
    movel([0.077659, -1.308677, -2.617895, -0.785818, 1.570796, 1.648455],accel_mss,speed_ms,0,blend_radius_m)
    movel([0.077187, -1.309039, -2.617674, -0.785675, 1.570796, 1.647984],accel_mss,speed_ms,0,blend_radius_m)
    movel([0.076724, -1.309309, -2.617511, -0.785570, 1.570796, 1.647520],accel_mss,speed_ms,0,blend_radius_m)
    movel([0.076338, -1.309187, -2.617585, -0.785618, 1.570796, 1.647134],accel_mss,speed_ms,0,blend_radius_m)
    movel([0.076209, -1.308628, -2.617924, -0.785837, 1.570796, 1.647005],accel_mss,speed_ms,0,blend_radius_m)
    movel([0.076116, -1.307960, -2.618330, -0.786100, 1.570796, 1.646913],accel_mss,speed_ms,0,blend_radius_m)
    movel([0.076083, -1.307280, -2.618742, -0.786368, 1.570796, 1.646879],accel_mss,speed_ms,0,blend_radius_m)
    movel([0.076095, -1.306774, -2.619048, -0.786567, 1.570796, 1.646891],accel_mss,speed_ms,0,blend_radius_m)
    movel([0.076142, -1.306449, -2.619244, -0.786696, 1.570796, 1.646938],accel_mss,speed_ms,0,blend_radius_m)
    movel([0.076248, -1.306149, -2.619426, -0.786815, 1.570796, 1.647044],accel_mss,speed_ms,0,blend_radius_m)
    movel([0.076446, -1.305763, -2.619659, -0.786968, 1.570796, 1.647243],accel_mss,speed_ms,0,blend_radius_m)
    movel([0.076797, -1.305253, -2.619966, -0.787170, 1.570796, 1.647593],accel_mss,speed_ms,0,blend_radius_m)
    movel([0.077222, -1.304834, -2.620218, -0.787337, 1.570796, 1.648018],accel_mss,speed_ms,0,blend_radius_m)
    movel([0.077828, -1.304417, -2.620470, -0.787503, 1.570796, 1.648625],accel_mss,speed_ms,0,blend_radius_m)
    movel([0.078794, -1.303880, -2.620792, -0.787717, 1.570796, 1.649591],accel_mss,speed_ms,0,blend_radius_m)
    movel([0.080203, -1.303163, -2.621223, -0.788003, 1.570796, 1.651000],accel_mss,speed_ms,0,blend_radius_m)
    movel([0.081785, -1.302416, -2.621671, -0.788302, 1.570796, 1.652581],accel_mss,speed_ms,0,blend_radius_m)
    movel([0.083247, -1.301763, -2.622062, -0.788564, 1.570796, 1.654043],accel_mss,speed_ms,0,blend_radius_m)
    movel([0.084162, -1.301411, -2.622272, -0.788706, 1.570796, 1.654958],accel_mss,speed_ms,0,blend_radius_m)
    movel([0.084675, -1.301251, -2.622368, -0.788770, 1.570796, 1.655472],accel_mss,speed_ms,0,blend_radius_m)
    movel([0.084988, -1.301189, -2.622405, -0.788795, 1.570796, 1.655784],accel_mss,speed_ms,0,blend_radius_m)
    movel([0.085477, -1.301278, -2.622352, -0.788759, 1.570796, 1.656273],accel_mss,speed_ms,0,blend_radius_m)
    movel([0.085801, -1.301477, -2.622233, -0.788679, 1.570796, 1.656597],accel_mss,speed_ms,0,blend_radius_m)
    movel([0.086025, -1.301709, -2.622094, -0.788586, 1.570796, 1.656822],accel_mss,speed_ms,0,blend_radius_m)
    movel([0.086213, -1.302208, -2.621795, -0.788386, 1.570796, 1.657010],accel_mss,speed_ms,0,blend_radius_m)
    movel([0.086374, -1.303118, -2.621250, -0.788021, 1.570796, 1.657170],accel_mss,speed_ms,0,blend_radius_m)
    movel([0.086472, -1.304054, -2.620688, -0.787647, 1.570796, 1.657269],accel_mss,speed_ms,0,blend_radius_m)
    movel([0.086421, -1.304572, -2.620376, -0.787441, 1.570796, 1.657218],accel_mss,speed_ms,0,blend_radius_m)
    speed_ms = 0.003
    movel([0.086236, -1.308210, -2.621895, -0.782283, 1.570796, 1.657033],accel_mss,speed_ms,0,blend_radius_m)
    speed_ms = 0.007
    movel([0.085836, -1.308401, -2.621780, -0.782208, 1.570796, 1.656632],accel_mss,speed_ms,0,blend_radius_m)
    movel([0.085399, -1.308529, -2.621702, -0.782158, 1.570796, 1.656196],accel_mss,speed_ms,0,blend_radius_m)
    movel([0.085110, -1.308423, -2.621767, -0.782199, 1.570796, 1.655906],accel_mss,speed_ms,0,blend_radius_m)
    movel([0.085056, -1.308187, -2.621909, -0.782292, 1.570796, 1.655852],accel_mss,speed_ms,0,blend_radius_m)
    movel([0.085010, -1.307895, -2.622086, -0.782408, 1.570796, 1.655807],accel_mss,speed_ms,0,blend_radius_m)
    movel([0.084978, -1.307569, -2.622283, -0.782537, 1.570796, 1.655775],accel_mss,speed_ms,0,blend_radius_m)
    movel([0.084892, -1.306955, -2.622654, -0.782780, 1.570796, 1.655688],accel_mss,speed_ms,0,blend_radius_m)
    movel([0.084735, -1.306571, -2.622886, -0.782932, 1.570796, 1.655531],accel_mss,speed_ms,0,blend_radius_m)
    movel([0.084474, -1.306352, -2.623017, -0.783019, 1.570796, 1.655271],accel_mss,speed_ms,0,blend_radius_m)
    movel([0.084085, -1.306251, -2.623078, -0.783059, 1.570796, 1.654882],accel_mss,speed_ms,0,blend_radius_m)
    movel([0.083756, -1.306270, -2.623067, -0.783052, 1.570796, 1.654553],accel_mss,speed_ms,0,blend_radius_m)
    movel([0.083385, -1.306376, -2.623003, -0.783010, 1.570796, 1.654181],accel_mss,speed_ms,0,blend_radius_m)
    movel([0.082789, -1.306629, -2.622851, -0.782910, 1.570796, 1.653585],accel_mss,speed_ms,0,blend_radius_m)
    movel([0.081437, -1.307268, -2.622465, -0.782656, 1.570796, 1.652233],accel_mss,speed_ms,0,blend_radius_m)
    movel([0.079639, -1.308139, -2.621939, -0.782312, 1.570796, 1.650435],accel_mss,speed_ms,0,blend_radius_m)
    movel([0.078834, -1.308575, -2.621675, -0.782140, 1.570796, 1.649630],accel_mss,speed_ms,0,blend_radius_m)
    movel([0.078346, -1.308923, -2.621464, -0.782002, 1.570796, 1.649142],accel_mss,speed_ms,0,blend_radius_m)
    movel([0.077948, -1.309333, -2.621215, -0.781841, 1.570796, 1.648744],accel_mss,speed_ms,0,blend_radius_m)
    movel([0.077690, -1.309749, -2.620962, -0.781677, 1.570796, 1.648486],accel_mss,speed_ms,0,blend_radius_m)
    movel([0.077544, -1.310200, -2.620689, -0.781500, 1.570796, 1.648340],accel_mss,speed_ms,0,blend_radius_m)
    movel([0.077508, -1.310694, -2.620388, -0.781307, 1.570796, 1.648304],accel_mss,speed_ms,0,blend_radius_m)
    movel([0.077587, -1.311234, -2.620059, -0.781095, 1.570796, 1.648383],accel_mss,speed_ms,0,blend_radius_m)
    movel([0.077671, -1.311604, -2.619834, -0.780951, 1.570796, 1.648467],accel_mss,speed_ms,0,blend_radius_m)
    movel([0.077735, -1.311890, -2.619660, -0.780839, 1.570796, 1.648531],accel_mss,speed_ms,0,blend_radius_m)
    movel([0.077659, -1.312151, -2.619500, -0.780738, 1.570796, 1.648455],accel_mss,speed_ms,0,blend_radius_m)
    movel([0.077187, -1.312513, -2.619280, -0.780597, 1.570796, 1.647984],accel_mss,speed_ms,0,blend_radius_m)
    movel([0.076724, -1.312781, -2.619115, -0.780492, 1.570796, 1.647520],accel_mss,speed_ms,0,blend_radius_m)
    movel([0.076338, -1.312660, -2.619190, -0.780540, 1.570796, 1.647134],accel_mss,speed_ms,0,blend_radius_m)
    movel([0.076209, -1.312103, -2.619530, -0.780756, 1.570796, 1.647005],accel_mss,speed_ms,0,blend_radius_m)
    movel([0.076116, -1.311436, -2.619937, -0.781017, 1.570796, 1.646913],accel_mss,speed_ms,0,blend_radius_m)
    movel([0.076083, -1.310757, -2.620350, -0.781282, 1.570796, 1.646879],accel_mss,speed_ms,0,blend_radius_m)
    movel([0.076095, -1.310253, -2.620656, -0.781480, 1.570796, 1.646891],accel_mss,speed_ms,0,blend_radius_m)
    movel([0.076142, -1.309929, -2.620853, -0.781607, 1.570796, 1.646938],accel_mss,speed_ms,0,blend_radius_m)
    movel([0.076248, -1.309629, -2.621036, -0.781725, 1.570796, 1.647044],accel_mss,speed_ms,0,blend_radius_m)
    movel([0.076446, -1.309244, -2.621269, -0.781876, 1.570796, 1.647243],accel_mss,speed_ms,0,blend_radius_m)
    movel([0.076797, -1.308735, -2.621577, -0.782076, 1.570796, 1.647593],accel_mss,speed_ms,0,blend_radius_m)
    movel([0.077222, -1.308317, -2.621831, -0.782241, 1.570796, 1.648018],accel_mss,speed_ms,0,blend_radius_m)
    movel([0.077828, -1.307901, -2.622083, -0.782406, 1.570796, 1.648625],accel_mss,speed_ms,0,blend_radius_m)
    movel([0.078794, -1.307365, -2.622406, -0.782618, 1.570796, 1.649591],accel_mss,speed_ms,0,blend_radius_m)
    movel([0.080203, -1.306650, -2.622838, -0.782901, 1.570796, 1.651000],accel_mss,speed_ms,0,blend_radius_m)
    movel([0.081785, -1.305904, -2.623287, -0.783197, 1.570796, 1.652581],accel_mss,speed_ms,0,blend_radius_m)
    movel([0.083247, -1.305253, -2.623679, -0.783457, 1.570796, 1.654043],accel_mss,speed_ms,0,blend_radius_m)
    movel([0.084162, -1.304902, -2.623890, -0.783597, 1.570796, 1.654958],accel_mss,speed_ms,0,blend_radius_m)
    movel([0.084675, -1.304742, -2.623986, -0.783660, 1.570796, 1.655472],accel_mss,speed_ms,0,blend_radius_m)
    movel([0.084988, -1.304680, -2.624023, -0.783685, 1.570796, 1.655784],accel_mss,speed_ms,0,blend_radius_m)
    movel([0.085477, -1.304770, -2.623970, -0.783650, 1.570796, 1.656273],accel_mss,speed_ms,0,blend_radius_m)
    movel([0.085801, -1.304968, -2.623851, -0.783571, 1.570796, 1.656597],accel_mss,speed_ms,0,blend_radius_m)
    movel([0.086025, -1.305199, -2.623712, -0.783478, 1.570796, 1.656822],accel_mss,speed_ms,0,blend_radius_m)
    movel([0.086213, -1.305697, -2.623412, -0.783280, 1.570796, 1.657010],accel_mss,speed_ms,0,blend_radius_m)
    movel([0.086374, -1.306605, -2.622865, -0.782919, 1.570796, 1.657170],accel_mss,speed_ms,0,blend_radius_m)
    movel([0.086472, -1.307539, -2.622301, -0.782549, 1.570796, 1.657269],accel_mss,speed_ms,0,blend_radius_m)
    movel([0.086421, -1.308056, -2.621989, -0.782344, 1.570796, 1.657218],accel_mss,speed_ms,0,blend_radius_m)
    speed_ms = 0.003
    movel([0.086236, -1.294441, -2.615396, -0.802552, 1.570796, 1.657033],accel_mss,speed_ms,0,blend_radius_m)
    speed_ms = 1.000
    movel([0.086236, -1.268202, -2.602010, -0.842178, 1.570796, 1.657033],accel_mss,speed_ms,0,blend_radius_m)
    movel([0.090839, -1.274742, -2.598244, -0.839403, 1.570796, 1.661635],accel_mss,speed_ms,0,blend_radius_m)
    movel([0.090839, -1.300888, -2.611545, -0.799956, 1.570796, 1.661635],accel_mss,speed_ms,0,blend_radius_m)
    speed_ms = 0.003
    movel([0.090839, -1.311132, -2.616400, -0.784857, 1.570796, 1.661635],accel_mss,speed_ms,0,blend_radius_m)
    speed_ms = 0.007
    movel([0.091231, -1.310851, -2.616572, -0.784967, 1.570796, 1.662027],accel_mss,speed_ms,0,blend_radius_m)
    movel([0.093076, -1.310222, -2.616955, -0.785212, 1.570796, 1.663872],accel_mss,speed_ms,0,blend_radius_m)
    movel([0.094912, -1.309640, -2.617309, -0.785440, 1.570796, 1.665708],accel_mss,speed_ms,0,blend_radius_m)
    movel([0.095311, -1.309662, -2.617295, -0.785431, 1.570796, 1.666108],accel_mss,speed_ms,0,blend_radius_m)
    movel([0.095304, -1.309901, -2.617150, -0.785338, 1.570796, 1.666100],accel_mss,speed_ms,0,blend_radius_m)
    movel([0.094896, -1.310250, -2.616938, -0.785201, 1.570796, 1.665692],accel_mss,speed_ms,0,blend_radius_m)
    movel([0.094536, -1.310423, -2.616832, -0.785134, 1.570796, 1.665332],accel_mss,speed_ms,0,blend_radius_m)
    movel([0.093961, -1.310638, -2.616701, -0.785050, 1.570796, 1.664758],accel_mss,speed_ms,0,blend_radius_m)
    movel([0.092892, -1.310989, -2.616487, -0.784913, 1.570796, 1.663688],accel_mss,speed_ms,0,blend_radius_m)
    movel([0.091876, -1.311310, -2.616291, -0.784788, 1.570796, 1.662673],accel_mss,speed_ms,0,blend_radius_m)
    movel([0.091309, -1.311465, -2.616196, -0.784727, 1.570796, 1.662105],accel_mss,speed_ms,0,blend_radius_m)
    movel([0.090961, -1.311529, -2.616157, -0.784703, 1.570796, 1.661757],accel_mss,speed_ms,0,blend_radius_m)
    movel([0.090736, -1.311417, -2.616225, -0.784746, 1.570796, 1.661532],accel_mss,speed_ms,0,blend_radius_m)
    movel([0.090839, -1.311132, -2.616400, -0.784857, 1.570796, 1.661635],accel_mss,speed_ms,0,blend_radius_m)
    speed_ms = 0.003
    movel([0.090839, -1.314601, -2.618001, -0.779787, 1.570796, 1.661635],accel_mss,speed_ms,0,blend_radius_m)
    speed_ms = 0.007
    movel([0.091231, -1.314320, -2.618174, -0.779896, 1.570796, 1.662027],accel_mss,speed_ms,0,blend_radius_m)
    movel([0.093076, -1.313693, -2.618558, -0.780138, 1.570796, 1.663872],accel_mss,speed_ms,0,blend_radius_m)
    movel([0.094912, -1.313112, -2.618913, -0.780364, 1.570796, 1.665708],accel_mss,speed_ms,0,blend_radius_m)
    movel([0.095311, -1.313135, -2.618899, -0.780355, 1.570796, 1.666108],accel_mss,speed_ms,0,blend_radius_m)
    movel([0.095304, -1.313373, -2.618754, -0.780263, 1.570796, 1.666100],accel_mss,speed_ms,0,blend_radius_m)
    movel([0.094896, -1.313720, -2.618541, -0.780128, 1.570796, 1.665692],accel_mss,speed_ms,0,blend_radius_m)
    movel([0.094536, -1.313893, -2.618435, -0.780061, 1.570796, 1.665332],accel_mss,speed_ms,0,blend_radius_m)
    movel([0.093961, -1.314108, -2.618304, -0.779978, 1.570796, 1.664758],accel_mss,speed_ms,0,blend_radius_m)
    movel([0.092892, -1.314458, -2.618089, -0.779842, 1.570796, 1.663688],accel_mss,speed_ms,0,blend_radius_m)
    movel([0.091876, -1.314778, -2.617893, -0.779719, 1.570796, 1.662673],accel_mss,speed_ms,0,blend_radius_m)
    movel([0.091309, -1.314933, -2.617797, -0.779659, 1.570796, 1.662105],accel_mss,speed_ms,0,blend_radius_m)
    movel([0.090961, -1.314997, -2.617758, -0.779634, 1.570796, 1.661757],accel_mss,speed_ms,0,blend_radius_m)
    movel([0.090736, -1.314885, -2.617826, -0.779677, 1.570796, 1.661532],accel_mss,speed_ms,0,blend_radius_m)
    movel([0.090839, -1.314601, -2.618001, -0.779787, 1.570796, 1.661635],accel_mss,speed_ms,0,blend_radius_m)
    speed_ms = 0.003
    movel([0.090839, -1.300888, -2.611545, -0.799956, 1.570796, 1.661635],accel_mss,speed_ms,0,blend_radius_m)
    speed_ms = 1.000
    movel([0.090839, -1.274742, -2.598244, -0.839403, 1.570796, 1.661635],accel_mss,speed_ms,0,blend_radius_m)
    movel([0.090283, -1.274574, -2.598342, -0.839473, 1.570796, 1.661079],accel_mss,speed_ms,0,blend_radius_m)
    movel([0.090283, -1.300723, -2.611644, -0.800022, 1.570796, 1.661079],accel_mss,speed_ms,0,blend_radius_m)
    speed_ms = 0.003
    movel([0.090283, -1.310968, -2.616500, -0.784921, 1.570796, 1.661079],accel_mss,speed_ms,0,blend_radius_m)
    speed_ms = 0.007
    movel([0.091304, -1.309341, -2.617491, -0.785557, 1.570796, 1.662100],accel_mss,speed_ms,0,blend_radius_m)
    movel([0.091772, -1.308890, -2.617765, -0.785734, 1.570796, 1.662568],accel_mss,speed_ms,0,blend_radius_m)
    movel([0.092217, -1.308558, -2.617967, -0.785864, 1.570796, 1.663014],accel_mss,speed_ms,0,blend_radius_m)
    movel([0.092713, -1.308300, -2.618123, -0.785966, 1.570796, 1.663510],accel_mss,speed_ms,0,blend_radius_m)
    movel([0.093344, -1.308063, -2.618267, -0.786059, 1.570796, 1.664141],accel_mss,speed_ms,0,blend_radius_m)
    movel([0.094712, -1.307930, -2.618348, -0.786111, 1.570796, 1.665509],accel_mss,speed_ms,0,blend_radius_m)
    movel([0.095678, -1.308467, -2.618022, -0.785900, 1.570796, 1.666474],accel_mss,speed_ms,0,blend_radius_m)
    movel([0.096003, -1.309536, -2.617373, -0.785481, 1.570796, 1.666799],accel_mss,speed_ms,0,blend_radius_m)
    movel([0.095606, -1.310869, -2.616560, -0.784960, 1.570796, 1.666402],accel_mss,speed_ms,0,blend_radius_m)
    movel([0.095281, -1.311375, -2.616251, -0.784763, 1.570796, 1.666077],accel_mss,speed_ms,0,blend_radius_m)
    movel([0.094834, -1.311913, -2.615923, -0.784553, 1.570796, 1.665631],accel_mss,speed_ms,0,blend_radius_m)
    movel([0.094350, -1.312398, -2.615626, -0.784365, 1.570796, 1.665146],accel_mss,speed_ms,0,blend_radius_m)
    movel([0.093908, -1.312733, -2.615421, -0.784235, 1.570796, 1.664704],accel_mss,speed_ms,0,blend_radius_m)
    movel([0.093410, -1.312978, -2.615271, -0.784140, 1.570796, 1.664206],accel_mss,speed_ms,0,blend_radius_m)
    movel([0.093084, -1.313110, -2.615190, -0.784089, 1.570796, 1.663881],accel_mss,speed_ms,0,blend_radius_m)
    movel([0.092771, -1.313220, -2.615122, -0.784047, 1.570796, 1.663568],accel_mss,speed_ms,0,blend_radius_m)
    movel([0.091175, -1.313300, -2.615073, -0.784016, 1.570796, 1.661972],accel_mss,speed_ms,0,blend_radius_m)
    movel([0.090238, -1.312456, -2.615591, -0.784343, 1.570796, 1.661034],accel_mss,speed_ms,0,blend_radius_m)
    movel([0.090283, -1.310968, -2.616500, -0.784921, 1.570796, 1.661079],accel_mss,speed_ms,0,blend_radius_m)
    speed_ms = 0.003
    movel([0.090283, -1.314437, -2.618102, -0.779850, 1.570796, 1.661079],accel_mss,speed_ms,0,blend_radius_m)
    speed_ms = 0.007
    movel([0.091304, -1.312814, -2.619095, -0.780479, 1.570796, 1.662100],accel_mss,speed_ms,0,blend_radius_m)
    movel([0.091772, -1.312364, -2.619370, -0.780654, 1.570796, 1.662568],accel_mss,speed_ms,0,blend_radius_m)
    movel([0.092217, -1.312033, -2.619573, -0.780784, 1.570796, 1.663014],accel_mss,speed_ms,0,blend_radius_m)
    movel([0.092713, -1.311775, -2.619730, -0.780884, 1.570796, 1.663510],accel_mss,speed_ms,0,blend_radius_m)
    movel([0.093344, -1.311539, -2.619874, -0.780976, 1.570796, 1.664141],accel_mss,speed_ms,0,blend_radius_m)
    movel([0.094712, -1.311406, -2.619954, -0.781028, 1.570796, 1.665509],accel_mss,speed_ms,0,blend_radius_m)
    movel([0.095678, -1.311942, -2.619628, -0.780819, 1.570796, 1.666474],accel_mss,speed_ms,0,blend_radius_m)
    movel([0.096003, -1.313008, -2.618977, -0.780404, 1.570796, 1.666799],accel_mss,speed_ms,0,blend_radius_m)
    movel([0.095606, -1.314338, -2.618162, -0.779889, 1.570796, 1.666402],accel_mss,speed_ms,0,blend_radius_m)
    movel([0.095281, -1.314843, -2.617852, -0.779693, 1.570796, 1.666077],accel_mss,speed_ms,0,blend_radius_m)
    movel([0.094834, -1.315380, -2.617523, -0.779486, 1.570796, 1.665631],accel_mss,speed_ms,0,blend_radius_m)
    movel([0.094350, -1.315864, -2.617225, -0.779300, 1.570796, 1.665146],accel_mss,speed_ms,0,blend_radius_m)
    movel([0.093908, -1.316198, -2.617019, -0.779171, 1.570796, 1.664704],accel_mss,speed_ms,0,blend_radius_m)
    movel([0.093410, -1.316443, -2.616869, -0.779078, 1.570796, 1.664206],accel_mss,speed_ms,0,blend_radius_m)
    movel([0.093084, -1.316574, -2.616788, -0.779027, 1.570796, 1.663881],accel_mss,speed_ms,0,blend_radius_m)
    movel([0.092771, -1.316684, -2.616720, -0.778985, 1.570796, 1.663568],accel_mss,speed_ms,0,blend_radius_m)
    movel([0.091175, -1.316764, -2.616671, -0.778954, 1.570796, 1.661972],accel_mss,speed_ms,0,blend_radius_m)
    movel([0.090238, -1.315921, -2.617190, -0.779278, 1.570796, 1.661034],accel_mss,speed_ms,0,blend_radius_m)
    movel([0.090283, -1.314437, -2.618102, -0.779850, 1.570796, 1.661079],accel_mss,speed_ms,0,blend_radius_m)
    speed_ms = 0.003
    movel([0.090283, -1.300723, -2.611644, -0.800022, 1.570796, 1.661079],accel_mss,speed_ms,0,blend_radius_m)
    speed_ms = 1.000
    movel([0.090283, -1.274574, -2.598342, -0.839473, 1.570796, 1.661079],accel_mss,speed_ms,0,blend_radius_m)
    movel([0.090194, -1.273895, -2.598735, -0.839759, 1.570796, 1.660990],accel_mss,speed_ms,0,blend_radius_m)
    movel([0.090194, -1.300054, -2.612046, -0.800289, 1.570796, 1.660990],accel_mss,speed_ms,0,blend_radius_m)
    speed_ms = 0.003
    movel([0.090194, -1.310304, -2.616905, -0.785180, 1.570796, 1.660990],accel_mss,speed_ms,0,blend_radius_m)
    speed_ms = 0.007
    movel([0.091881, -1.308449, -2.618033, -0.785907, 1.570796, 1.662678],accel_mss,speed_ms,0,blend_radius_m)
    movel([0.093261, -1.307710, -2.618481, -0.786198, 1.570796, 1.664057],accel_mss,speed_ms,0,blend_radius_m)
    movel([0.094545, -1.307450, -2.618639, -0.786300, 1.570796, 1.665342],accel_mss,speed_ms,0,blend_radius_m)
    movel([0.095586, -1.307711, -2.618480, -0.786197, 1.570796, 1.666383],accel_mss,speed_ms,0,blend_radius_m)
    movel([0.096268, -1.308456, -2.618029, -0.785904, 1.570796, 1.667065],accel_mss,speed_ms,0,blend_radius_m)
    movel([0.096402, -1.308965, -2.617719, -0.785704, 1.570796, 1.667198],accel_mss,speed_ms,0,blend_radius_m)
    movel([0.096383, -1.309618, -2.617323, -0.785449, 1.570796, 1.667179],accel_mss,speed_ms,0,blend_radius_m)
    movel([0.096219, -1.310326, -2.616892, -0.785172, 1.570796, 1.667015],accel_mss,speed_ms,0,blend_radius_m)
    movel([0.095924, -1.311003, -2.616479, -0.784908, 1.570796, 1.666721],accel_mss,speed_ms,0,blend_radius_m)
    movel([0.095337, -1.311867, -2.615950, -0.784571, 1.570796, 1.666134],accel_mss,speed_ms,0,blend_radius_m)
    movel([0.094603, -1.312601, -2.615502, -0.784287, 1.570796, 1.665399],accel_mss,speed_ms,0,blend_radius_m)
    movel([0.093731, -1.313184, -2.615144, -0.784061, 1.570796, 1.664527],accel_mss,speed_ms,0,blend_radius_m)
    movel([0.092744, -1.313607, -2.614885, -0.783897, 1.570796, 1.663540],accel_mss,speed_ms,0,blend_radius_m)
    movel([0.090757, -1.313624, -2.614874, -0.783890, 1.570796, 1.661553],accel_mss,speed_ms,0,blend_radius_m)
    movel([0.089757, -1.312332, -2.615666, -0.784391, 1.570796, 1.660553],accel_mss,speed_ms,0,blend_radius_m)
    movel([0.090194, -1.310304, -2.616905, -0.785180, 1.570796, 1.660990],accel_mss,speed_ms,0,blend_radius_m)
    speed_ms = 0.003
    movel([0.090194, -1.313774, -2.618508, -0.780107, 1.570796, 1.660990],accel_mss,speed_ms,0,blend_radius_m)
    speed_ms = 0.007
    movel([0.091881, -1.311924, -2.619639, -0.780826, 1.570796, 1.662678],accel_mss,speed_ms,0,blend_radius_m)
    movel([0.093261, -1.311186, -2.620089, -0.781114, 1.570796, 1.664057],accel_mss,speed_ms,0,blend_radius_m)
    movel([0.094545, -1.310927, -2.620246, -0.781215, 1.570796, 1.665342],accel_mss,speed_ms,0,blend_radius_m)
    movel([0.095586, -1.311188, -2.620088, -0.781113, 1.570796, 1.666383],accel_mss,speed_ms,0,blend_radius_m)
    movel([0.096268, -1.311931, -2.619635, -0.780823, 1.570796, 1.667065],accel_mss,speed_ms,0,blend_radius_m)
    movel([0.096402, -1.312439, -2.619325, -0.780625, 1.570796, 1.667198],accel_mss,speed_ms,0,blend_radius_m)
    movel([0.096383, -1.313090, -2.618927, -0.780372, 1.570796, 1.667179],accel_mss,speed_ms,0,blend_radius_m)
    movel([0.096219, -1.313796, -2.618494, -0.780098, 1.570796, 1.667015],accel_mss,speed_ms,0,blend_radius_m)
    movel([0.095924, -1.314472, -2.618080, -0.779837, 1.570796, 1.666721],accel_mss,speed_ms,0,blend_radius_m)
    movel([0.095337, -1.315334, -2.617551, -0.779504, 1.570796, 1.666134],accel_mss,speed_ms,0,blend_radius_m)
    movel([0.094603, -1.316066, -2.617101, -0.779222, 1.570796, 1.665399],accel_mss,speed_ms,0,blend_radius_m)
    movel([0.093731, -1.316648, -2.616742, -0.778999, 1.570796, 1.664527],accel_mss,speed_ms,0,blend_radius_m)
    movel([0.092744, -1.317070, -2.616482, -0.778837, 1.570796, 1.663540],accel_mss,speed_ms,0,blend_radius_m)
    movel([0.090757, -1.317087, -2.616472, -0.778830, 1.570796, 1.661553],accel_mss,speed_ms,0,blend_radius_m)
    movel([0.089757, -1.315798, -2.617265, -0.779325, 1.570796, 1.660553],accel_mss,speed_ms,0,blend_radius_m)
    movel([0.090194, -1.313774, -2.618508, -0.780107, 1.570796, 1.660990],accel_mss,speed_ms,0,blend_radius_m)
    speed_ms = 0.003
    movel([0.090194, -1.300054, -2.612046, -0.800289, 1.570796, 1.660990],accel_mss,speed_ms,0,blend_radius_m)
    speed_ms = 1.000
    movel([0.090194, -1.273895, -2.598735, -0.839759, 1.570796, 1.660990],accel_mss,speed_ms,0,blend_radius_m)
    movel([0.074648, -1.283142, -2.593332, -0.835915, 1.570796, 1.645444],accel_mss,speed_ms,0,blend_radius_m)
    movel([0.074648, -1.309165, -2.606523, -0.796701, 1.570796, 1.645444],accel_mss,speed_ms,0,blend_radius_m)
    speed_ms = 0.003
    movel([0.074648, -1.319355, -2.611336, -0.781699, 1.570796, 1.645444],accel_mss,speed_ms,0,blend_radius_m)
    speed_ms = 0.007
    movel([0.074675, -1.319767, -2.611079, -0.781543, 1.570796, 1.645472],accel_mss,speed_ms,0,blend_radius_m)
    movel([0.074553, -1.320280, -2.610760, -0.781349, 1.570796, 1.645349],accel_mss,speed_ms,0,blend_radius_m)
